   1:  PR[GP1:91,1] = PR[GP1:90,1] + 21.012;
   1:  PR[GP1:91,2] = PR[GP1:90,2] + -18.046;
   1:L PR[91] 10mm/sec CNT100;
   1:  PR[GP1:91,1] = PR[GP1:90,1] + 21.989;
   1:  PR[GP1:91,2] = PR[GP1:90,2] + -17.133;
   1:L PR[91] 10mm/sec CNT100;
   1:  PR[GP1:91,1] = PR[GP1:90,1] + 23.164;
   1:  PR[GP1:91,2] = PR[GP1:90,2] + -15.934;
   1:L PR[91] 10mm/sec CNT100;
   1:  PR[GP1:91,1] = PR[GP1:90,1] + 23.554;
   1:  PR[GP1:91,2] = PR[GP1:90,2] + -15.432;
   1:L PR[91] 10mm/sec CNT100;
   1:  PR[GP1:91,1] = PR[GP1:90,1] + 24.718;
   1:  PR[GP1:91,2] = PR[GP1:90,2] + -13.798;
   1:L PR[91] 10mm/sec CNT100;
   1:  PR[GP1:91,1] = PR[GP1:90,1] + 24.953;
   1:  PR[GP1:91,2] = PR[GP1:90,2] + -13.491;
   1:L PR[91] 10mm/sec CNT100;
   1:  PR[GP1:91,1] = PR[GP1:90,1] + 26.370;
   1:  PR[GP1:91,2] = PR[GP1:90,2] + -10.907;
   1:L PR[91] 10mm/sec CNT100;
   1:  PR[GP1:91,1] = PR[GP1:90,1] + 27.373;
   1:  PR[GP1:91,2] = PR[GP1:90,2] + -8.158;
   1:L PR[91] 10mm/sec CNT100;
   1:  PR[GP1:91,1] = PR[GP1:90,1] + 27.934;
   1:  PR[GP1:91,2] = PR[GP1:90,2] + -5.322;
   1:L PR[91] 10mm/sec CNT100;
   1:  PR[GP1:91,1] = PR[GP1:90,1] + 28.066;
   1:  PR[GP1:91,2] = PR[GP1:90,2] + -2.515;
   1:L PR[91] 10mm/sec CNT100;
   1:  PR[GP1:91,1] = PR[GP1:90,1] + 27.956;
   1:  PR[GP1:91,2] = PR[GP1:90,2] + -1.536;
   1:L PR[91] 10mm/sec CNT100;
   1:  PR[GP1:91,1] = PR[GP1:90,1] + 27.632;
   1:  PR[GP1:91,2] = PR[GP1:90,2] + 0.969;
   1:L PR[91] 10mm/sec CNT100;
   1:  PR[GP1:91,1] = PR[GP1:90,1] + 26.516;
   1:  PR[GP1:91,2] = PR[GP1:90,2] + 4.243;
   1:L PR[91] 10mm/sec CNT100;
   1:  PR[GP1:91,1] = PR[GP1:90,1] + 24.774;
   1:  PR[GP1:91,2] = PR[GP1:90,2] + 7.177;
   1:L PR[91] 10mm/sec CNT100;
   1:  PR[GP1:91,1] = PR[GP1:90,1] + 22.490;
   1:  PR[GP1:91,2] = PR[GP1:90,2] + 9.677;
   1:L PR[91] 10mm/sec CNT100;
   1:  PR[GP1:91,1] = PR[GP1:90,1] + 21.756;
   1:  PR[GP1:91,2] = PR[GP1:90,2] + 10.214;
   1:L PR[91] 10mm/sec CNT100;
   1:  PR[GP1:91,1] = PR[GP1:90,1] + 19.758;
   1:  PR[GP1:91,2] = PR[GP1:90,2] + 11.659;
   1:L PR[91] 10mm/sec CNT100;
   1:  PR[GP1:91,1] = PR[GP1:90,1] + 16.663;
   1:  PR[GP1:91,2] = PR[GP1:90,2] + 13.071;
   1:L PR[91] 10mm/sec CNT100;
   1:  PR[GP1:91,1] = PR[GP1:90,1] + 13.308;
   1:  PR[GP1:91,2] = PR[GP1:90,2] + 13.868;
   1:L PR[91] 10mm/sec CNT100;
   1:  PR[GP1:91,1] = PR[GP1:90,1] + 9.910;
   1:  PR[GP1:91,2] = PR[GP1:90,2] + 14.002;
   1:L PR[91] 10mm/sec CNT100;
   1:  PR[GP1:91,1] = PR[GP1:90,1] + 6.569;
   1:  PR[GP1:91,2] = PR[GP1:90,2] + 13.484;
   1:L PR[91] 10mm/sec CNT100;
   1:  PR[GP1:91,1] = PR[GP1:90,1] + 3.289;
   1:  PR[GP1:91,2] = PR[GP1:90,2] + 12.332;
   1:L PR[91] 10mm/sec CNT100;
   1:  PR[GP1:91,1] = PR[GP1:90,1] + 2.867;
   1:  PR[GP1:91,2] = PR[GP1:90,2] + 12.167;
   1:L PR[91] 10mm/sec CNT100;
   1:  PR[GP1:91,1] = PR[GP1:90,1] + 2.443;
   1:  PR[GP1:91,2] = PR[GP1:90,2] + 11.963;
   1:L PR[91] 10mm/sec CNT100;
   1:  PR[GP1:91,1] = PR[GP1:90,1] + 1.134;
   1:  PR[GP1:91,2] = PR[GP1:90,2] + 11.701;
   1:L PR[91] 10mm/sec CNT100;
   1:  PR[GP1:91,1] = PR[GP1:90,1] + 0.392;
   1:  PR[GP1:91,2] = PR[GP1:90,2] + 11.851;
   1:L PR[91] 10mm/sec CNT100;
   1:  PR[GP1:91,1] = PR[GP1:90,1] + -0.582;
   1:  PR[GP1:91,2] = PR[GP1:90,2] + 12.179;
   1:L PR[91] 10mm/sec CNT100;
   1:  PR[GP1:91,1] = PR[GP1:90,1] + -1.398;
   1:  PR[GP1:91,2] = PR[GP1:90,2] + 12.423;
   1:L PR[91] 10mm/sec CNT100;
   1:  PR[GP1:91,1] = PR[GP1:90,1] + -1.769;
   1:  PR[GP1:91,2] = PR[GP1:90,2] + 12.518;
   1:L PR[91] 10mm/sec CNT100;
   1:  PR[GP1:91,1] = PR[GP1:90,1] + -4.247;
   1:  PR[GP1:91,2] = PR[GP1:90,2] + 13.099;
   1:L PR[91] 10mm/sec CNT100;
   1:  PR[GP1:91,1] = PR[GP1:90,1] + -5.225;
   1:  PR[GP1:91,2] = PR[GP1:90,2] + 13.264;
   1:L PR[91] 10mm/sec CNT100;
   1:  PR[GP1:91,1] = PR[GP1:90,1] + -7.861;
   1:  PR[GP1:91,2] = PR[GP1:90,2] + 13.602;
   1:L PR[91] 10mm/sec CNT100;
   1:  PR[GP1:91,1] = PR[GP1:90,1] + -10.489;
   1:  PR[GP1:91,2] = PR[GP1:90,2] + 13.626;
   1:L PR[91] 10mm/sec CNT100;
   1:  PR[GP1:91,1] = PR[GP1:90,1] + -11.733;
   1:  PR[GP1:91,2] = PR[GP1:90,2] + 13.530;
   1:L PR[91] 10mm/sec CNT100;
   1:  PR[GP1:91,1] = PR[GP1:90,1] + -13.508;
   1:  PR[GP1:91,2] = PR[GP1:90,2] + 13.328;
   1:L PR[91] 10mm/sec CNT100;
   1:  PR[GP1:91,1] = PR[GP1:90,1] + -17.046;
   1:  PR[GP1:91,2] = PR[GP1:90,2] + 12.458;
   1:L PR[91] 10mm/sec CNT100;
   1:  PR[GP1:91,1] = PR[GP1:90,1] + -17.326;
   1:  PR[GP1:91,2] = PR[GP1:90,2] + 12.351;
   1:L PR[91] 10mm/sec CNT100;
   1:  PR[GP1:91,1] = PR[GP1:90,1] + -18.942;
   1:  PR[GP1:91,2] = PR[GP1:90,2] + 11.624;
   1:L PR[91] 10mm/sec CNT100;
   1:  PR[GP1:91,1] = PR[GP1:90,1] + -20.346;
   1:  PR[GP1:91,2] = PR[GP1:90,2] + 10.955;
   1:L PR[91] 10mm/sec CNT100;
   1:  PR[GP1:91,1] = PR[GP1:90,1] + -20.668;
   1:  PR[GP1:91,2] = PR[GP1:90,2] + 10.742;
   1:L PR[91] 10mm/sec CNT100;
   1:  PR[GP1:91,1] = PR[GP1:90,1] + -23.016;
   1:  PR[GP1:91,2] = PR[GP1:90,2] + 8.981;
   1:L PR[91] 10mm/sec CNT100;
   1:  PR[GP1:91,1] = PR[GP1:90,1] + -23.744;
   1:  PR[GP1:91,2] = PR[GP1:90,2] + 8.223;
   1:L PR[91] 10mm/sec CNT100;
   1:  PR[GP1:91,1] = PR[GP1:90,1] + -25.239;
   1:  PR[GP1:91,2] = PR[GP1:90,2] + 6.489;
   1:L PR[91] 10mm/sec CNT100;
   1:  PR[GP1:91,1] = PR[GP1:90,1] + -25.974;
   1:  PR[GP1:91,2] = PR[GP1:90,2] + 5.258;
   1:L PR[91] 10mm/sec CNT100;
   1:  PR[GP1:91,1] = PR[GP1:90,1] + -26.895;
   1:  PR[GP1:91,2] = PR[GP1:90,2] + 3.561;
   1:L PR[91] 10mm/sec CNT100;
   1:  PR[GP1:91,1] = PR[GP1:90,1] + -27.389;
   1:  PR[GP1:91,2] = PR[GP1:90,2] + 2.055;
   1:L PR[91] 10mm/sec CNT100;
   1:  PR[GP1:91,1] = PR[GP1:90,1] + -27.899;
   1:  PR[GP1:91,2] = PR[GP1:90,2] + 0.349;
   1:L PR[91] 10mm/sec CNT100;
   1:  PR[GP1:91,1] = PR[GP1:90,1] + -27.981;
   1:  PR[GP1:91,2] = PR[GP1:90,2] + -1.199;
   1:L PR[91] 10mm/sec CNT100;
   1:  PR[GP1:91,1] = PR[GP1:90,1] + -28.107;
   1:  PR[GP1:91,2] = PR[GP1:90,2] + -2.353;
   1:L PR[91] 10mm/sec CNT100;
   1:  PR[GP1:91,1] = PR[GP1:90,1] + -28.126;
   1:  PR[GP1:91,2] = PR[GP1:90,2] + -3.024;
   1:L PR[91] 10mm/sec CNT100;
   1:  PR[GP1:91,1] = PR[GP1:90,1] + -27.809;
   1:  PR[GP1:91,2] = PR[GP1:90,2] + -4.338;
   1:L PR[91] 10mm/sec CNT100;
   1:  PR[GP1:91,1] = PR[GP1:90,1] + -27.384;
   1:  PR[GP1:91,2] = PR[GP1:90,2] + -6.573;
   1:L PR[91] 10mm/sec CNT100;
   1:  PR[GP1:91,1] = PR[GP1:90,1] + -26.082;
   1:  PR[GP1:91,2] = PR[GP1:90,2] + -9.859;
   1:L PR[91] 10mm/sec CNT100;
   1:  PR[GP1:91,1] = PR[GP1:90,1] + -25.098;
   1:  PR[GP1:91,2] = PR[GP1:90,2] + -11.325;
   1:L PR[91] 10mm/sec CNT100;
   1:  PR[GP1:91,1] = PR[GP1:90,1] + -24.065;
   1:  PR[GP1:91,2] = PR[GP1:90,2] + -12.765;
   1:L PR[91] 10mm/sec CNT100;
   1:  PR[GP1:91,1] = PR[GP1:90,1] + -23.826;
   1:  PR[GP1:91,2] = PR[GP1:90,2] + -13.037;
   1:L PR[91] 10mm/sec CNT100;
   1:  PR[GP1:91,1] = PR[GP1:90,1] + -21.725;
   1:  PR[GP1:91,2] = PR[GP1:90,2] + -15.036;
   1:L PR[91] 10mm/sec CNT100;
   1:  PR[GP1:91,1] = PR[GP1:90,1] + -19.832;
   1:  PR[GP1:91,2] = PR[GP1:90,2] + -16.187;
   1:  PR[GP1:91,3] = PR[GP1:90,3] + 37.400;
   1:L PR[91] 10mm/sec CNT100;
   1:  PR[GP1:91,1] = PR[GP1:90,1] + -19.095;
   1:  PR[GP1:91,2] = PR[GP1:90,2] + -16.677;
   1:L PR[91] 10mm/sec CNT100;
   1:  PR[GP1:91,1] = PR[GP1:90,1] + -16.804;
   1:  PR[GP1:91,2] = PR[GP1:90,2] + -18.166;
   1:L PR[91] 10mm/sec CNT100;
   1:  PR[GP1:91,1] = PR[GP1:90,1] + -14.134;
   1:  PR[GP1:91,2] = PR[GP1:90,2] + -19.465;
   1:L PR[91] 10mm/sec CNT100;
   1:  PR[GP1:91,1] = PR[GP1:90,1] + -13.059;
   1:  PR[GP1:91,2] = PR[GP1:90,2] + -19.937;
   1:L PR[91] 10mm/sec CNT100;
   1:  PR[GP1:91,1] = PR[GP1:90,1] + -10.699;
   1:  PR[GP1:91,2] = PR[GP1:90,2] + -20.757;
   1:L PR[91] 10mm/sec CNT100;
   1:  PR[GP1:91,1] = PR[GP1:90,1] + -8.029;
   1:  PR[GP1:91,2] = PR[GP1:90,2] + -21.395;
   1:L PR[91] 10mm/sec CNT100;
   1:  PR[GP1:91,1] = PR[GP1:90,1] + -6.377;
   1:  PR[GP1:91,2] = PR[GP1:90,2] + -21.749;
   1:L PR[91] 10mm/sec CNT100;
   1:  PR[GP1:91,1] = PR[GP1:90,1] + -5.286;
   1:  PR[GP1:91,2] = PR[GP1:90,2] + -21.845;
   1:L PR[91] 10mm/sec CNT100;
   1:  PR[GP1:91,1] = PR[GP1:90,1] + -1.083;
   1:  PR[GP1:91,2] = PR[GP1:90,2] + -22.066;
   1:L PR[91] 10mm/sec CNT100;
   1:  PR[GP1:91,1] = PR[GP1:90,1] + -0.849;
   1:  PR[GP1:91,2] = PR[GP1:90,2] + -22.058;
   1:L PR[91] 10mm/sec CNT100;
   1:  PR[GP1:91,1] = PR[GP1:90,1] + 0.695;
   1:  PR[GP1:91,2] = PR[GP1:90,2] + -21.837;
   1:L PR[91] 10mm/sec CNT100;
   1:  PR[GP1:91,1] = PR[GP1:90,1] + 3.686;
   1:  PR[GP1:91,2] = PR[GP1:90,2] + -21.563;
   1:L PR[91] 10mm/sec CNT100;
   1:  PR[GP1:91,1] = PR[GP1:90,1] + 4.828;
   1:  PR[GP1:91,2] = PR[GP1:90,2] + -21.636;
   1:L PR[91] 10mm/sec CNT100;
   1:  PR[GP1:91,1] = PR[GP1:90,1] + 7.253;
   1:  PR[GP1:91,2] = PR[GP1:90,2] + -22.196;
   1:L PR[91] 10mm/sec CNT100;
   1:  PR[GP1:91,1] = PR[GP1:90,1] + 7.750;
   1:  PR[GP1:91,2] = PR[GP1:90,2] + -22.271;
   1:L PR[91] 10mm/sec CNT100;
   1:  PR[GP1:91,1] = PR[GP1:90,1] + 9.996;
   1:  PR[GP1:91,2] = PR[GP1:90,2] + -22.414;
   1:L PR[91] 10mm/sec CNT100;
   1:  PR[GP1:91,1] = PR[GP1:90,1] + 10.580;
   1:  PR[GP1:91,2] = PR[GP1:90,2] + -22.410;
   1:L PR[91] 10mm/sec CNT100;
   1:  PR[GP1:91,1] = PR[GP1:90,1] + 12.766;
   1:  PR[GP1:91,2] = PR[GP1:90,2] + -22.182;
   1:L PR[91] 10mm/sec CNT100;
   1:  PR[GP1:91,1] = PR[GP1:90,1] + 13.348;
   1:  PR[GP1:91,2] = PR[GP1:90,2] + -22.084;
   1:L PR[91] 10mm/sec CNT100;
   1:  PR[GP1:91,1] = PR[GP1:90,1] + 15.521;
   1:  PR[GP1:91,2] = PR[GP1:90,2] + -21.475;
   1:L PR[91] 10mm/sec CNT100;
   1:  PR[GP1:91,1] = PR[GP1:90,1] + 15.993;
   1:  PR[GP1:91,2] = PR[GP1:90,2] + -21.316;
   1:L PR[91] 10mm/sec CNT100;
   1:  PR[GP1:91,1] = PR[GP1:90,1] + 18.220;
   1:  PR[GP1:91,2] = PR[GP1:90,2] + -20.263;
   1:L PR[91] 10mm/sec CNT100;
   1:  PR[GP1:91,1] = PR[GP1:90,1] + 18.464;
   1:  PR[GP1:91,2] = PR[GP1:90,2] + -20.135;
   1:L PR[91] 10mm/sec CNT100;
   1:  PR[GP1:91,1] = PR[GP1:90,1] + 20.758;
   1:  PR[GP1:91,2] = PR[GP1:90,2] + -18.540;
   1:L PR[91] 10mm/sec CNT100;
   1:  PR[GP1:91,1] = PR[GP1:90,1] + 22.565;
   1:  PR[GP1:91,2] = PR[GP1:90,2] + -16.852;
   1:L PR[91] 10mm/sec CNT100;
   1:  PR[GP1:91,1] = PR[GP1:90,1] + 22.942;
   1:  PR[GP1:91,2] = PR[GP1:90,2] + -16.467;
   1:L PR[91] 10mm/sec CNT100;
   1:  PR[GP1:91,1] = PR[GP1:90,1] + 24.069;
   1:  PR[GP1:91,2] = PR[GP1:90,2] + -15.016;
   1:L PR[91] 10mm/sec CNT100;
   1:  PR[GP1:91,1] = PR[GP1:90,1] + 24.767;
   1:  PR[GP1:91,2] = PR[GP1:90,2] + -14.036;
   1:L PR[91] 10mm/sec CNT100;
   1:  PR[GP1:91,1] = PR[GP1:90,1] + 25.287;
   1:  PR[GP1:91,2] = PR[GP1:90,2] + -13.094;
   1:L PR[91] 10mm/sec CNT100;
   1:  PR[GP1:91,1] = PR[GP1:90,1] + 26.166;
   1:  PR[GP1:91,2] = PR[GP1:90,2] + -11.348;
   1:L PR[91] 10mm/sec CNT100;
   1:  PR[GP1:91,1] = PR[GP1:90,1] + 26.521;
   1:  PR[GP1:91,2] = PR[GP1:90,2] + -10.307;
   1:L PR[91] 10mm/sec CNT100;
   1:  PR[GP1:91,1] = PR[GP1:90,1] + 27.176;
   1:  PR[GP1:91,2] = PR[GP1:90,2] + -8.541;
   1:L PR[91] 10mm/sec CNT100;
   1:  PR[GP1:91,1] = PR[GP1:90,1] + 27.757;
   1:  PR[GP1:91,2] = PR[GP1:90,2] + -5.709;
   1:L PR[91] 10mm/sec CNT100;
   1:  PR[GP1:91,1] = PR[GP1:90,1] + 27.820;
   1:  PR[GP1:91,2] = PR[GP1:90,2] + -3.864;
   1:L PR[91] 10mm/sec CNT100;
   1:  PR[GP1:91,1] = PR[GP1:90,1] + 27.835;
   1:  PR[GP1:91,2] = PR[GP1:90,2] + -2.835;
   1:L PR[91] 10mm/sec CNT100;
   1:  PR[GP1:91,1] = PR[GP1:90,1] + 27.396;
   1:  PR[GP1:91,2] = PR[GP1:90,2] + 0.695;
   1:L PR[91] 10mm/sec CNT100;
   1:  PR[GP1:91,1] = PR[GP1:90,1] + 26.293;
   1:  PR[GP1:91,2] = PR[GP1:90,2] + 3.983;
   1:L PR[91] 10mm/sec CNT100;
   1:  PR[GP1:91,1] = PR[GP1:90,1] + 24.552;
   1:  PR[GP1:91,2] = PR[GP1:90,2] + 6.933;
   1:L PR[91] 10mm/sec CNT100;
   1:  PR[GP1:91,1] = PR[GP1:90,1] + 22.263;
   1:  PR[GP1:91,2] = PR[GP1:90,2] + 9.449;
   1:L PR[91] 10mm/sec CNT100;
   1:  PR[GP1:91,1] = PR[GP1:90,1] + 20.511;
   1:  PR[GP1:91,2] = PR[GP1:90,2] + 10.732;
   1:L PR[91] 10mm/sec CNT100;
   1:  PR[GP1:91,1] = PR[GP1:90,1] + 19.522;
   1:  PR[GP1:91,2] = PR[GP1:90,2] + 11.448;
   1:L PR[91] 10mm/sec CNT100;
   1:  PR[GP1:91,1] = PR[GP1:90,1] + 16.409;
   1:  PR[GP1:91,2] = PR[GP1:90,2] + 12.874;
   1:L PR[91] 10mm/sec CNT100;
   1:  PR[GP1:91,1] = PR[GP1:90,1] + 13.155;
   1:  PR[GP1:91,2] = PR[GP1:90,2] + 13.652;
   1:L PR[91] 10mm/sec CNT100;
   1:  PR[GP1:91,1] = PR[GP1:90,1] + 9.719;
   1:  PR[GP1:91,2] = PR[GP1:90,2] + 13.804;
   1:L PR[91] 10mm/sec CNT100;
   1:  PR[GP1:91,1] = PR[GP1:90,1] + 9.011;
   1:  PR[GP1:91,2] = PR[GP1:90,2] + 13.706;
   1:L PR[91] 10mm/sec CNT100;
   1:  PR[GP1:91,1] = PR[GP1:90,1] + 6.398;
   1:  PR[GP1:91,2] = PR[GP1:90,2] + 13.292;
   1:L PR[91] 10mm/sec CNT100;
   1:  PR[GP1:91,1] = PR[GP1:90,1] + 3.118;
   1:  PR[GP1:91,2] = PR[GP1:90,2] + 12.148;
   1:L PR[91] 10mm/sec CNT100;
   1:  PR[GP1:91,1] = PR[GP1:90,1] + 2.622;
   1:  PR[GP1:91,2] = PR[GP1:90,2] + 11.953;
   1:L PR[91] 10mm/sec CNT100;
   1:  PR[GP1:91,1] = PR[GP1:90,1] + 1.327;
   1:  PR[GP1:91,2] = PR[GP1:90,2] + 11.705;
   1:L PR[91] 10mm/sec CNT100;
   1:  PR[GP1:91,1] = PR[GP1:90,1] + 0.669;
   1:  PR[GP1:91,2] = PR[GP1:90,2] + 11.858;
   1:L PR[91] 10mm/sec CNT100;
   1:  PR[GP1:91,1] = PR[GP1:90,1] + -0.435;
   1:  PR[GP1:91,2] = PR[GP1:90,2] + 12.188;
   1:L PR[91] 10mm/sec CNT100;
   1:  PR[GP1:91,1] = PR[GP1:90,1] + -0.928;
   1:  PR[GP1:91,2] = PR[GP1:90,2] + 12.315;
   1:L PR[91] 10mm/sec CNT100;
   1:  PR[GP1:91,1] = PR[GP1:90,1] + -2.534;
   1:  PR[GP1:91,2] = PR[GP1:90,2] + 12.694;
   1:L PR[91] 10mm/sec CNT100;
   1:  PR[GP1:91,1] = PR[GP1:90,1] + -3.060;
   1:  PR[GP1:91,2] = PR[GP1:90,2] + 12.812;
   1:L PR[91] 10mm/sec CNT100;
   1:  PR[GP1:91,1] = PR[GP1:90,1] + -4.631;
   1:  PR[GP1:91,2] = PR[GP1:90,2] + 13.077;
   1:L PR[91] 10mm/sec CNT100;
   1:  PR[GP1:91,1] = PR[GP1:90,1] + -6.914;
   1:  PR[GP1:91,2] = PR[GP1:90,2] + 13.369;
   1:L PR[91] 10mm/sec CNT100;
   1:  PR[GP1:91,1] = PR[GP1:90,1] + -10.028;
   1:  PR[GP1:91,2] = PR[GP1:90,2] + 13.428;
   1:L PR[91] 10mm/sec CNT100;
   1:  PR[GP1:91,1] = PR[GP1:90,1] + -12.823;
   1:  PR[GP1:91,2] = PR[GP1:90,2] + 13.118;
   1:L PR[91] 10mm/sec CNT100;
   1:  PR[GP1:91,1] = PR[GP1:90,1] + -16.123;
   1:  PR[GP1:91,2] = PR[GP1:90,2] + 12.304;
   1:L PR[91] 10mm/sec CNT100;
   1:  PR[GP1:91,1] = PR[GP1:90,1] + -16.912;
   1:  PR[GP1:91,2] = PR[GP1:90,2] + 12.003;
   1:L PR[91] 10mm/sec CNT100;
   1:  PR[GP1:91,1] = PR[GP1:90,1] + -19.663;
   1:  PR[GP1:91,2] = PR[GP1:90,2] + 10.766;
   1:L PR[91] 10mm/sec CNT100;
   1:  PR[GP1:91,1] = PR[GP1:90,1] + -19.823;
   1:  PR[GP1:91,2] = PR[GP1:90,2] + 10.679;
   1:L PR[91] 10mm/sec CNT100;
   1:  PR[GP1:91,1] = PR[GP1:90,1] + -20.996;
   1:  PR[GP1:91,2] = PR[GP1:90,2] + 9.844;
   1:L PR[91] 10mm/sec CNT100;
   1:  PR[GP1:91,1] = PR[GP1:90,1] + -22.533;
   1:  PR[GP1:91,2] = PR[GP1:90,2] + 8.692;
   1:L PR[91] 10mm/sec CNT100;
   1:  PR[GP1:91,1] = PR[GP1:90,1] + -22.765;
   1:  PR[GP1:91,2] = PR[GP1:90,2] + 8.450;
   1:L PR[91] 10mm/sec CNT100;
   1:  PR[GP1:91,1] = PR[GP1:90,1] + -24.701;
   1:  PR[GP1:91,2] = PR[GP1:90,2] + 6.205;
   1:L PR[91] 10mm/sec CNT100;
   1:  PR[GP1:91,1] = PR[GP1:90,1] + -25.091;
   1:  PR[GP1:91,2] = PR[GP1:90,2] + 5.551;
   1:L PR[91] 10mm/sec CNT100;
   1:  PR[GP1:91,1] = PR[GP1:90,1] + -26.314;
   1:  PR[GP1:91,2] = PR[GP1:90,2] + 3.296;
   1:L PR[91] 10mm/sec CNT100;
   1:  PR[GP1:91,1] = PR[GP1:90,1] + -26.610;
   1:  PR[GP1:91,2] = PR[GP1:90,2] + 2.395;
   1:L PR[91] 10mm/sec CNT100;
   1:  PR[GP1:91,1] = PR[GP1:90,1] + -27.292;
   1:  PR[GP1:91,2] = PR[GP1:90,2] + 0.114;
   1:L PR[91] 10mm/sec CNT100;
   1:  PR[GP1:91,1] = PR[GP1:90,1] + -27.342;
   1:  PR[GP1:91,2] = PR[GP1:90,2] + -0.825;
   1:L PR[91] 10mm/sec CNT100;
   1:  PR[GP1:91,1] = PR[GP1:90,1] + -27.420;
   1:  PR[GP1:91,2] = PR[GP1:90,2] + -1.538;
   1:L PR[91] 10mm/sec CNT100;
   1:  PR[GP1:91,1] = PR[GP1:90,1] + -27.467;
   1:  PR[GP1:91,2] = PR[GP1:90,2] + -3.238;
   1:L PR[91] 10mm/sec CNT100;
   1:  PR[GP1:91,1] = PR[GP1:90,1] + -27.297;
   1:  PR[GP1:91,2] = PR[GP1:90,2] + -3.942;
   1:L PR[91] 10mm/sec CNT100;
   1:  PR[GP1:91,1] = PR[GP1:90,1] + -26.763;
   1:  PR[GP1:91,2] = PR[GP1:90,2] + -6.745;
   1:L PR[91] 10mm/sec CNT100;
   1:  PR[GP1:91,1] = PR[GP1:90,1] + -25.976;
   1:  PR[GP1:91,2] = PR[GP1:90,2] + -8.742;
   1:L PR[91] 10mm/sec CNT100;
   1:  PR[GP1:91,1] = PR[GP1:90,1] + -25.440;
   1:  PR[GP1:91,2] = PR[GP1:90,2] + -9.977;
   1:L PR[91] 10mm/sec CNT100;
   1:  PR[GP1:91,1] = PR[GP1:90,1] + -25.345;
   1:  PR[GP1:91,2] = PR[GP1:90,2] + -10.127;
   1:L PR[91] 10mm/sec CNT100;
   1:  PR[GP1:91,1] = PR[GP1:90,1] + -23.474;
   1:  PR[GP1:91,2] = PR[GP1:90,2] + -12.733;
   1:L PR[91] 10mm/sec CNT100;
   1:  PR[GP1:91,1] = PR[GP1:90,1] + -22.802;
   1:  PR[GP1:91,2] = PR[GP1:90,2] + -13.499;
   1:L PR[91] 10mm/sec CNT100;
   1:  PR[GP1:91,1] = PR[GP1:90,1] + -21.280;
   1:  PR[GP1:91,2] = PR[GP1:90,2] + -14.947;
   1:L PR[91] 10mm/sec CNT100;
   1:  PR[GP1:91,1] = PR[GP1:90,1] + -18.916;
   1:  PR[GP1:91,2] = PR[GP1:90,2] + -16.501;
   1:  PR[GP1:91,3] = PR[GP1:90,3] + 38.500;
   1:L PR[91] 10mm/sec CNT100;
   1:  PR[GP1:91,1] = PR[GP1:90,1] + -15.891;
   1:  PR[GP1:91,2] = PR[GP1:90,2] + -18.471;
   1:L PR[91] 10mm/sec CNT100;
   1:  PR[GP1:91,1] = PR[GP1:90,1] + -13.552;
   1:  PR[GP1:91,2] = PR[GP1:90,2] + -19.609;
   1:L PR[91] 10mm/sec CNT100;
   1:  PR[GP1:91,1] = PR[GP1:90,1] + -11.911;
   1:  PR[GP1:91,2] = PR[GP1:90,2] + -20.329;
   1:L PR[91] 10mm/sec CNT100;
   1:  PR[GP1:91,1] = PR[GP1:90,1] + -9.976;
   1:  PR[GP1:91,2] = PR[GP1:90,2] + -21.001;
   1:L PR[91] 10mm/sec CNT100;
   1:  PR[GP1:91,1] = PR[GP1:90,1] + -6.564;
   1:  PR[GP1:91,2] = PR[GP1:90,2] + -21.817;
   1:L PR[91] 10mm/sec CNT100;
   1:  PR[GP1:91,1] = PR[GP1:90,1] + -5.457;
   1:  PR[GP1:91,2] = PR[GP1:90,2] + -22.054;
   1:L PR[91] 10mm/sec CNT100;
   1:  PR[GP1:91,1] = PR[GP1:90,1] + -4.733;
   1:  PR[GP1:91,2] = PR[GP1:90,2] + -22.118;
   1:L PR[91] 10mm/sec CNT100;
   1:  PR[GP1:91,1] = PR[GP1:90,1] + -0.660;
   1:  PR[GP1:91,2] = PR[GP1:90,2] + -22.332;
   1:L PR[91] 10mm/sec CNT100;
   1:  PR[GP1:91,1] = PR[GP1:90,1] + 0.067;
   1:  PR[GP1:91,2] = PR[GP1:90,2] + -22.399;
   1:L PR[91] 10mm/sec CNT100;
   1:  PR[GP1:91,1] = PR[GP1:90,1] + 4.181;
   1:  PR[GP1:91,2] = PR[GP1:90,2] + -22.017;
   1:L PR[91] 10mm/sec CNT100;
   1:  PR[GP1:91,1] = PR[GP1:90,1] + 5.247;
   1:  PR[GP1:91,2] = PR[GP1:90,2] + -22.084;
   1:L PR[91] 10mm/sec CNT100;
   1:  PR[GP1:91,1] = PR[GP1:90,1] + 6.980;
   1:  PR[GP1:91,2] = PR[GP1:90,2] + -22.475;
   1:L PR[91] 10mm/sec CNT100;
   1:  PR[GP1:91,1] = PR[GP1:90,1] + 8.189;
   1:  PR[GP1:91,2] = PR[GP1:90,2] + -22.656;
   1:L PR[91] 10mm/sec CNT100;
   1:  PR[GP1:91,1] = PR[GP1:90,1] + 9.649;
   1:  PR[GP1:91,2] = PR[GP1:90,2] + -22.750;
   1:L PR[91] 10mm/sec CNT100;
   1:  PR[GP1:91,1] = PR[GP1:90,1] + 11.005;
   1:  PR[GP1:91,2] = PR[GP1:90,2] + -22.739;
   1:L PR[91] 10mm/sec CNT100;
   1:  PR[GP1:91,1] = PR[GP1:90,1] + 12.338;
   1:  PR[GP1:91,2] = PR[GP1:90,2] + -22.600;
   1:L PR[91] 10mm/sec CNT100;
   1:  PR[GP1:91,1] = PR[GP1:90,1] + 13.748;
   1:  PR[GP1:91,2] = PR[GP1:90,2] + -22.364;
   1:L PR[91] 10mm/sec CNT100;
   1:  PR[GP1:91,1] = PR[GP1:90,1] + 15.010;
   1:  PR[GP1:91,2] = PR[GP1:90,2] + -22.010;
   1:L PR[91] 10mm/sec CNT100;
   1:  PR[GP1:91,1] = PR[GP1:90,1] + 16.359;
   1:  PR[GP1:91,2] = PR[GP1:90,2] + -21.556;
   1:L PR[91] 10mm/sec CNT100;
   1:  PR[GP1:91,1] = PR[GP1:90,1] + 17.629;
   1:  PR[GP1:91,2] = PR[GP1:90,2] + -20.956;
   1:L PR[91] 10mm/sec CNT100;
   1:  PR[GP1:91,1] = PR[GP1:90,1] + 18.786;
   1:  PR[GP1:91,2] = PR[GP1:90,2] + -20.350;
   1:L PR[91] 10mm/sec CNT100;
   1:  PR[GP1:91,1] = PR[GP1:90,1] + 20.151;
   1:  PR[GP1:91,2] = PR[GP1:90,2] + -19.396;
   1:L PR[91] 10mm/sec CNT100;
   1:  PR[GP1:91,1] = PR[GP1:90,1] + 20.988;
   1:  PR[GP1:91,2] = PR[GP1:90,2] + -18.773;
   1:L PR[91] 10mm/sec CNT100;
   1:  PR[GP1:91,1] = PR[GP1:90,1] + 22.521;
   1:  PR[GP1:91,2] = PR[GP1:90,2] + -17.270;
   1:L PR[91] 10mm/sec CNT100;
   1:  PR[GP1:91,1] = PR[GP1:90,1] + 22.928;
   1:  PR[GP1:91,2] = PR[GP1:90,2] + -16.854;
   1:L PR[91] 10mm/sec CNT100;
   1:  PR[GP1:91,1] = PR[GP1:90,1] + 24.594;
   1:  PR[GP1:91,2] = PR[GP1:90,2] + -14.584;
   1:L PR[91] 10mm/sec CNT100;
   1:  PR[GP1:91,1] = PR[GP1:90,1] + 25.711;
   1:  PR[GP1:91,2] = PR[GP1:90,2] + -12.559;
   1:L PR[91] 10mm/sec CNT100;
   1:  PR[GP1:91,1] = PR[GP1:90,1] + 26.045;
   1:  PR[GP1:91,2] = PR[GP1:90,2] + -11.895;
   1:L PR[91] 10mm/sec CNT100;
   1:  PR[GP1:91,1] = PR[GP1:90,1] + 26.567;
   1:  PR[GP1:91,2] = PR[GP1:90,2] + -10.480;
   1:L PR[91] 10mm/sec CNT100;
   1:  PR[GP1:91,1] = PR[GP1:90,1] + 27.047;
   1:  PR[GP1:91,2] = PR[GP1:90,2] + -9.029;
   1:L PR[91] 10mm/sec CNT100;
   1:  PR[GP1:91,1] = PR[GP1:90,1] + 27.183;
   1:  PR[GP1:91,2] = PR[GP1:90,2] + -8.364;
   1:L PR[91] 10mm/sec CNT100;
   1:  PR[GP1:91,1] = PR[GP1:90,1] + 27.582;
   1:  PR[GP1:91,2] = PR[GP1:90,2] + -6.102;
   1:L PR[91] 10mm/sec CNT100;
   1:  PR[GP1:91,1] = PR[GP1:90,1] + 27.694;
   1:  PR[GP1:91,2] = PR[GP1:90,2] + -3.225;
   1:L PR[91] 10mm/sec CNT100;
   1:  PR[GP1:91,1] = PR[GP1:90,1] + 27.195;
   1:  PR[GP1:91,2] = PR[GP1:90,2] + 0.389;
   1:L PR[91] 10mm/sec CNT100;
   1:  PR[GP1:91,1] = PR[GP1:90,1] + 26.701;
   1:  PR[GP1:91,2] = PR[GP1:90,2] + 1.818;
   1:L PR[91] 10mm/sec CNT100;
   1:  PR[GP1:91,1] = PR[GP1:90,1] + 26.070;
   1:  PR[GP1:91,2] = PR[GP1:90,2] + 3.722;
   1:L PR[91] 10mm/sec CNT100;
   1:  PR[GP1:91,1] = PR[GP1:90,1] + 24.330;
   1:  PR[GP1:91,2] = PR[GP1:90,2] + 6.689;
   1:L PR[91] 10mm/sec CNT100;
   1:  PR[GP1:91,1] = PR[GP1:90,1] + 22.035;
   1:  PR[GP1:91,2] = PR[GP1:90,2] + 9.222;
   1:L PR[91] 10mm/sec CNT100;
   1:  PR[GP1:91,1] = PR[GP1:90,1] + 19.282;
   1:  PR[GP1:91,2] = PR[GP1:90,2] + 11.237;
   1:L PR[91] 10mm/sec CNT100;
   1:  PR[GP1:91,1] = PR[GP1:90,1] + 16.261;
   1:  PR[GP1:91,2] = PR[GP1:90,2] + 12.645;
   1:L PR[91] 10mm/sec CNT100;
   1:  PR[GP1:91,1] = PR[GP1:90,1] + 13.003;
   1:  PR[GP1:91,2] = PR[GP1:90,2] + 13.436;
   1:L PR[91] 10mm/sec CNT100;
   1:  PR[GP1:91,1] = PR[GP1:90,1] + 9.620;
   1:  PR[GP1:91,2] = PR[GP1:90,2] + 13.586;
   1:L PR[91] 10mm/sec CNT100;
   1:  PR[GP1:91,1] = PR[GP1:90,1] + 7.086;
   1:  PR[GP1:91,2] = PR[GP1:90,2] + 13.236;
   1:L PR[91] 10mm/sec CNT100;
   1:  PR[GP1:91,1] = PR[GP1:90,1] + 6.226;
   1:  PR[GP1:91,2] = PR[GP1:90,2] + 13.099;
   1:L PR[91] 10mm/sec CNT100;
   1:  PR[GP1:91,1] = PR[GP1:90,1] + 2.820;
   1:  PR[GP1:91,2] = PR[GP1:90,2] + 11.916;
   1:L PR[91] 10mm/sec CNT100;
   1:  PR[GP1:91,1] = PR[GP1:90,1] + 1.538;
   1:  PR[GP1:91,2] = PR[GP1:90,2] + 11.705;
   1:L PR[91] 10mm/sec CNT100;
   1:  PR[GP1:91,1] = PR[GP1:90,1] + 0.971;
   1:  PR[GP1:91,2] = PR[GP1:90,2] + 11.821;
   1:L PR[91] 10mm/sec CNT100;
   1:  PR[GP1:91,1] = PR[GP1:90,1] + 0.528;
   1:  PR[GP1:91,2] = PR[GP1:90,2] + 11.954;
   1:L PR[91] 10mm/sec CNT100;
   1:  PR[GP1:91,1] = PR[GP1:90,1] + -0.085;
   1:  PR[GP1:91,2] = PR[GP1:90,2] + 12.112;
   1:L PR[91] 10mm/sec CNT100;
   1:  PR[GP1:91,1] = PR[GP1:90,1] + -1.879;
   1:  PR[GP1:91,2] = PR[GP1:90,2] + 12.527;
   1:L PR[91] 10mm/sec CNT100;
   1:  PR[GP1:91,1] = PR[GP1:90,1] + -4.037;
   1:  PR[GP1:91,2] = PR[GP1:90,2] + 12.890;
   1:L PR[91] 10mm/sec CNT100;
   1:  PR[GP1:91,1] = PR[GP1:90,1] + -5.962;
   1:  PR[GP1:91,2] = PR[GP1:90,2] + 13.137;
   1:L PR[91] 10mm/sec CNT100;
   1:  PR[GP1:91,1] = PR[GP1:90,1] + -9.327;
   1:  PR[GP1:91,2] = PR[GP1:90,2] + 13.196;
   1:L PR[91] 10mm/sec CNT100;
   1:  PR[GP1:91,1] = PR[GP1:90,1] + -11.088;
   1:  PR[GP1:91,2] = PR[GP1:90,2] + 13.026;
   1:L PR[91] 10mm/sec CNT100;
   1:  PR[GP1:91,1] = PR[GP1:90,1] + -12.136;
   1:  PR[GP1:91,2] = PR[GP1:90,2] + 12.908;
   1:L PR[91] 10mm/sec CNT100;
   1:  PR[GP1:91,1] = PR[GP1:90,1] + -15.201;
   1:  PR[GP1:91,2] = PR[GP1:90,2] + 12.151;
   1:L PR[91] 10mm/sec CNT100;
   1:  PR[GP1:91,1] = PR[GP1:90,1] + -16.498;
   1:  PR[GP1:91,2] = PR[GP1:90,2] + 11.656;
   1:L PR[91] 10mm/sec CNT100;
   1:  PR[GP1:91,1] = PR[GP1:90,1] + -18.532;
   1:  PR[GP1:91,2] = PR[GP1:90,2] + 10.741;
   1:L PR[91] 10mm/sec CNT100;
   1:  PR[GP1:91,1] = PR[GP1:90,1] + -19.213;
   1:  PR[GP1:91,2] = PR[GP1:90,2] + 10.369;
   1:L PR[91] 10mm/sec CNT100;
   1:  PR[GP1:91,1] = PR[GP1:90,1] + -21.917;
   1:  PR[GP1:91,2] = PR[GP1:90,2] + 8.438;
   1:L PR[91] 10mm/sec CNT100;
   1:  PR[GP1:91,1] = PR[GP1:90,1] + -23.406;
   1:  PR[GP1:91,2] = PR[GP1:90,2] + 6.799;
   1:L PR[91] 10mm/sec CNT100;
   1:  PR[GP1:91,1] = PR[GP1:90,1] + -24.162;
   1:  PR[GP1:91,2] = PR[GP1:90,2] + 5.922;
   1:L PR[91] 10mm/sec CNT100;
   1:  PR[GP1:91,1] = PR[GP1:90,1] + -24.209;
   1:  PR[GP1:91,2] = PR[GP1:90,2] + 5.844;
   1:L PR[91] 10mm/sec CNT100;
   1:  PR[GP1:91,1] = PR[GP1:90,1] + -25.730;
   1:  PR[GP1:91,2] = PR[GP1:90,2] + 3.038;
   1:L PR[91] 10mm/sec CNT100;
   1:  PR[GP1:91,1] = PR[GP1:90,1] + -26.688;
   1:  PR[GP1:91,2] = PR[GP1:90,2] + -0.131;
   1:L PR[91] 10mm/sec CNT100;
   1:  PR[GP1:91,1] = PR[GP1:90,1] + -26.732;
   1:  PR[GP1:91,2] = PR[GP1:90,2] + -0.713;
   1:L PR[91] 10mm/sec CNT100;
   1:  PR[GP1:91,1] = PR[GP1:90,1] + -26.807;
   1:  PR[GP1:91,2] = PR[GP1:90,2] + -3.452;
   1:L PR[91] 10mm/sec CNT100;
   1:  PR[GP1:91,1] = PR[GP1:90,1] + -26.785;
   1:  PR[GP1:91,2] = PR[GP1:90,2] + -3.546;
   1:L PR[91] 10mm/sec CNT100;
   1:  PR[GP1:91,1] = PR[GP1:90,1] + -26.546;
   1:  PR[GP1:91,2] = PR[GP1:90,2] + -4.800;
   1:L PR[91] 10mm/sec CNT100;
   1:  PR[GP1:91,1] = PR[GP1:90,1] + -26.118;
   1:  PR[GP1:91,2] = PR[GP1:90,2] + -6.738;
   1:L PR[91] 10mm/sec CNT100;
   1:  PR[GP1:91,1] = PR[GP1:90,1] + -26.078;
   1:  PR[GP1:91,2] = PR[GP1:90,2] + -6.912;
   1:L PR[91] 10mm/sec CNT100;
   1:  PR[GP1:91,1] = PR[GP1:90,1] + -25.995;
   1:  PR[GP1:91,2] = PR[GP1:90,2] + -7.118;
   1:L PR[91] 10mm/sec CNT100;
   1:  PR[GP1:91,1] = PR[GP1:90,1] + -24.719;
   1:  PR[GP1:91,2] = PR[GP1:90,2] + -10.057;
   1:L PR[91] 10mm/sec CNT100;
   1:  PR[GP1:91,1] = PR[GP1:90,1] + -24.274;
   1:  PR[GP1:91,2] = PR[GP1:90,2] + -10.764;
   1:L PR[91] 10mm/sec CNT100;
   1:  PR[GP1:91,1] = PR[GP1:90,1] + -22.883;
   1:  PR[GP1:91,2] = PR[GP1:90,2] + -12.701;
   1:L PR[91] 10mm/sec CNT100;
   1:  PR[GP1:91,1] = PR[GP1:90,1] + -21.778;
   1:  PR[GP1:91,2] = PR[GP1:90,2] + -13.961;
   1:L PR[91] 10mm/sec CNT100;
   1:  PR[GP1:91,1] = PR[GP1:90,1] + -20.834;
   1:  PR[GP1:91,2] = PR[GP1:90,2] + -14.858;
   1:L PR[91] 10mm/sec CNT100;
   1:  PR[GP1:91,1] = PR[GP1:90,1] + -20.389;
   1:  PR[GP1:91,2] = PR[GP1:90,2] + -14.770;
   1:  PR[GP1:91,3] = PR[GP1:90,3] + 39.600;
   1:L PR[91] 10mm/sec CNT100;
   1:  PR[GP1:91,1] = PR[GP1:90,1] + -18.113;
   1:  PR[GP1:91,2] = PR[GP1:90,2] + -16.722;
   1:L PR[91] 10mm/sec CNT100;
   1:  PR[GP1:91,1] = PR[GP1:90,1] + -17.695;
   1:  PR[GP1:91,2] = PR[GP1:90,2] + -17.008;
   1:L PR[91] 10mm/sec CNT100;
   1:  PR[GP1:91,1] = PR[GP1:90,1] + -14.979;
   1:  PR[GP1:91,2] = PR[GP1:90,2] + -18.775;
   1:L PR[91] 10mm/sec CNT100;
   1:  PR[GP1:91,1] = PR[GP1:90,1] + -12.969;
   1:  PR[GP1:91,2] = PR[GP1:90,2] + -19.753;
   1:L PR[91] 10mm/sec CNT100;
   1:  PR[GP1:91,1] = PR[GP1:90,1] + -10.762;
   1:  PR[GP1:91,2] = PR[GP1:90,2] + -20.721;
   1:L PR[91] 10mm/sec CNT100;
   1:  PR[GP1:91,1] = PR[GP1:90,1] + -9.253;
   1:  PR[GP1:91,2] = PR[GP1:90,2] + -21.245;
   1:L PR[91] 10mm/sec CNT100;
   1:  PR[GP1:91,1] = PR[GP1:90,1] + -5.099;
   1:  PR[GP1:91,2] = PR[GP1:90,2] + -22.239;
   1:L PR[91] 10mm/sec CNT100;
   1:  PR[GP1:91,1] = PR[GP1:90,1] + -4.537;
   1:  PR[GP1:91,2] = PR[GP1:90,2] + -22.359;
   1:L PR[91] 10mm/sec CNT100;
   1:  PR[GP1:91,1] = PR[GP1:90,1] + -4.179;
   1:  PR[GP1:91,2] = PR[GP1:90,2] + -22.390;
   1:L PR[91] 10mm/sec CNT100;
   1:  PR[GP1:91,1] = PR[GP1:90,1] + -2.024;
   1:  PR[GP1:91,2] = PR[GP1:90,2] + -22.504;
   1:L PR[91] 10mm/sec CNT100;
   1:  PR[GP1:91,1] = PR[GP1:90,1] + 0.476;
   1:  PR[GP1:91,2] = PR[GP1:90,2] + -22.773;
   1:L PR[91] 10mm/sec CNT100;
   1:  PR[GP1:91,1] = PR[GP1:90,1] + 1.191;
   1:  PR[GP1:91,2] = PR[GP1:90,2] + -22.803;
   1:L PR[91] 10mm/sec CNT100;
   1:  PR[GP1:91,1] = PR[GP1:90,1] + 4.701;
   1:  PR[GP1:91,2] = PR[GP1:90,2] + -22.468;
   1:L PR[91] 10mm/sec CNT100;
   1:  PR[GP1:91,1] = PR[GP1:90,1] + 5.689;
   1:  PR[GP1:91,2] = PR[GP1:90,2] + -22.529;
   1:L PR[91] 10mm/sec CNT100;
   1:  PR[GP1:91,1] = PR[GP1:90,1] + 6.707;
   1:  PR[GP1:91,2] = PR[GP1:90,2] + -22.753;
   1:L PR[91] 10mm/sec CNT100;
   1:  PR[GP1:91,1] = PR[GP1:90,1] + 8.628;
   1:  PR[GP1:91,2] = PR[GP1:90,2] + -23.042;
   1:L PR[91] 10mm/sec CNT100;
   1:  PR[GP1:91,1] = PR[GP1:90,1] + 9.302;
   1:  PR[GP1:91,2] = PR[GP1:90,2] + -23.085;
   1:L PR[91] 10mm/sec CNT100;
   1:  PR[GP1:91,1] = PR[GP1:90,1] + 11.431;
   1:  PR[GP1:91,2] = PR[GP1:90,2] + -23.069;
   1:L PR[91] 10mm/sec CNT100;
   1:  PR[GP1:91,1] = PR[GP1:90,1] + 11.909;
   1:  PR[GP1:91,2] = PR[GP1:90,2] + -23.019;
   1:L PR[91] 10mm/sec CNT100;
   1:  PR[GP1:91,1] = PR[GP1:90,1] + 14.149;
   1:  PR[GP1:91,2] = PR[GP1:90,2] + -22.644;
   1:L PR[91] 10mm/sec CNT100;
   1:  PR[GP1:91,1] = PR[GP1:90,1] + 14.498;
   1:  PR[GP1:91,2] = PR[GP1:90,2] + -22.546;
   1:L PR[91] 10mm/sec CNT100;
   1:  PR[GP1:91,1] = PR[GP1:90,1] + 16.724;
   1:  PR[GP1:91,2] = PR[GP1:90,2] + -21.797;
   1:L PR[91] 10mm/sec CNT100;
   1:  PR[GP1:91,1] = PR[GP1:90,1] + 17.037;
   1:  PR[GP1:91,2] = PR[GP1:90,2] + -21.649;
   1:L PR[91] 10mm/sec CNT100;
   1:  PR[GP1:91,1] = PR[GP1:90,1] + 19.108;
   1:  PR[GP1:91,2] = PR[GP1:90,2] + -20.564;
   1:L PR[91] 10mm/sec CNT100;
   1:  PR[GP1:91,1] = PR[GP1:90,1] + 19.493;
   1:  PR[GP1:91,2] = PR[GP1:90,2] + -20.296;
   1:L PR[91] 10mm/sec CNT100;
   1:  PR[GP1:91,1] = PR[GP1:90,1] + 21.261;
   1:  PR[GP1:91,2] = PR[GP1:90,2] + -18.978;
   1:L PR[91] 10mm/sec CNT100;
   1:  PR[GP1:91,1] = PR[GP1:90,1] + 21.821;
   1:  PR[GP1:91,2] = PR[GP1:90,2] + -18.429;
   1:L PR[91] 10mm/sec CNT100;
   1:  PR[GP1:91,1] = PR[GP1:90,1] + 23.148;
   1:  PR[GP1:91,2] = PR[GP1:90,2] + -17.072;
   1:L PR[91] 10mm/sec CNT100;
   1:  PR[GP1:91,1] = PR[GP1:90,1] + 24.741;
   1:  PR[GP1:91,2] = PR[GP1:90,2] + -14.860;
   1:L PR[91] 10mm/sec CNT100;
   1:  PR[GP1:91,1] = PR[GP1:90,1] + 26.007;
   1:  PR[GP1:91,2] = PR[GP1:90,2] + -12.369;
   1:L PR[91] 10mm/sec CNT100;
   1:  PR[GP1:91,1] = PR[GP1:90,1] + 26.508;
   1:  PR[GP1:91,2] = PR[GP1:90,2] + -10.856;
   1:L PR[91] 10mm/sec CNT100;
   1:  PR[GP1:91,1] = PR[GP1:90,1] + 26.878;
   1:  PR[GP1:91,2] = PR[GP1:90,2] + -9.854;
   1:L PR[91] 10mm/sec CNT100;
   1:  PR[GP1:91,1] = PR[GP1:90,1] + 26.972;
   1:  PR[GP1:91,2] = PR[GP1:90,2] + -9.569;
   1:L PR[91] 10mm/sec CNT100;
   1:  PR[GP1:91,1] = PR[GP1:90,1] + 27.357;
   1:  PR[GP1:91,2] = PR[GP1:90,2] + -7.683;
   1:L PR[91] 10mm/sec CNT100;
   1:  PR[GP1:91,1] = PR[GP1:90,1] + 27.543;
   1:  PR[GP1:91,2] = PR[GP1:90,2] + -6.613;
   1:L PR[91] 10mm/sec CNT100;
   1:  PR[GP1:91,1] = PR[GP1:90,1] + 27.604;
   1:  PR[GP1:91,2] = PR[GP1:90,2] + -3.657;
   1:L PR[91] 10mm/sec CNT100;
   1:  PR[GP1:91,1] = PR[GP1:90,1] + 27.454;
   1:  PR[GP1:91,2] = PR[GP1:90,2] + -2.655;
   1:L PR[91] 10mm/sec CNT100;
   1:  PR[GP1:91,1] = PR[GP1:90,1] + 27.109;
   1:  PR[GP1:91,2] = PR[GP1:90,2] + 0.004;
   1:L PR[91] 10mm/sec CNT100;
   1:  PR[GP1:91,1] = PR[GP1:90,1] + 26.463;
   1:  PR[GP1:91,2] = PR[GP1:90,2] + 1.876;
   1:L PR[91] 10mm/sec CNT100;
   1:  PR[GP1:91,1] = PR[GP1:90,1] + 25.962;
   1:  PR[GP1:91,2] = PR[GP1:90,2] + 3.394;
   1:L PR[91] 10mm/sec CNT100;
   1:  PR[GP1:91,1] = PR[GP1:90,1] + 25.530;
   1:  PR[GP1:91,2] = PR[GP1:90,2] + 4.150;
   1:L PR[91] 10mm/sec CNT100;
   1:  PR[GP1:91,1] = PR[GP1:90,1] + 24.196;
   1:  PR[GP1:91,2] = PR[GP1:90,2] + 6.402;
   1:L PR[91] 10mm/sec CNT100;
   1:  PR[GP1:91,1] = PR[GP1:90,1] + 21.906;
   1:  PR[GP1:91,2] = PR[GP1:90,2] + 8.955;
   1:L PR[91] 10mm/sec CNT100;
   1:  PR[GP1:91,1] = PR[GP1:90,1] + 19.193;
   1:  PR[GP1:91,2] = PR[GP1:90,2] + 10.974;
   1:L PR[91] 10mm/sec CNT100;
   1:  PR[GP1:91,1] = PR[GP1:90,1] + 18.194;
   1:  PR[GP1:91,2] = PR[GP1:90,2] + 11.453;
   1:L PR[91] 10mm/sec CNT100;
   1:  PR[GP1:91,1] = PR[GP1:90,1] + 16.157;
   1:  PR[GP1:91,2] = PR[GP1:90,2] + 12.403;
   1:L PR[91] 10mm/sec CNT100;
   1:  PR[GP1:91,1] = PR[GP1:90,1] + 12.851;
   1:  PR[GP1:91,2] = PR[GP1:90,2] + 13.219;
   1:L PR[91] 10mm/sec CNT100;
   1:  PR[GP1:91,1] = PR[GP1:90,1] + 9.521;
   1:  PR[GP1:91,2] = PR[GP1:90,2] + 13.369;
   1:L PR[91] 10mm/sec CNT100;
   1:  PR[GP1:91,1] = PR[GP1:90,1] + 6.108;
   1:  PR[GP1:91,2] = PR[GP1:90,2] + 12.889;
   1:L PR[91] 10mm/sec CNT100;
   1:  PR[GP1:91,1] = PR[GP1:90,1] + 4.989;
   1:  PR[GP1:91,2] = PR[GP1:90,2] + 12.530;
   1:L PR[91] 10mm/sec CNT100;
   1:  PR[GP1:91,1] = PR[GP1:90,1] + 3.048;
   1:  PR[GP1:91,2] = PR[GP1:90,2] + 11.857;
   1:L PR[91] 10mm/sec CNT100;
   1:  PR[GP1:91,1] = PR[GP1:90,1] + 1.753;
   1:  PR[GP1:91,2] = PR[GP1:90,2] + 11.664;
   1:L PR[91] 10mm/sec CNT100;
   1:  PR[GP1:91,1] = PR[GP1:90,1] + -0.697;
   1:  PR[GP1:91,2] = PR[GP1:90,2] + 12.241;
   1:L PR[91] 10mm/sec CNT100;
   1:  PR[GP1:91,1] = PR[GP1:90,1] + -3.443;
   1:  PR[GP1:91,2] = PR[GP1:90,2] + 12.703;
   1:L PR[91] 10mm/sec CNT100;
   1:  PR[GP1:91,1] = PR[GP1:90,1] + -5.012;
   1:  PR[GP1:91,2] = PR[GP1:90,2] + 12.904;
   1:L PR[91] 10mm/sec CNT100;
   1:  PR[GP1:91,1] = PR[GP1:90,1] + -7.309;
   1:  PR[GP1:91,2] = PR[GP1:90,2] + 12.950;
   1:L PR[91] 10mm/sec CNT100;
   1:  PR[GP1:91,1] = PR[GP1:90,1] + -8.564;
   1:  PR[GP1:91,2] = PR[GP1:90,2] + 12.957;
   1:L PR[91] 10mm/sec CNT100;
   1:  PR[GP1:91,1] = PR[GP1:90,1] + -11.248;
   1:  PR[GP1:91,2] = PR[GP1:90,2] + 12.698;
   1:L PR[91] 10mm/sec CNT100;
   1:  PR[GP1:91,1] = PR[GP1:90,1] + -11.480;
   1:  PR[GP1:91,2] = PR[GP1:90,2] + 12.660;
   1:L PR[91] 10mm/sec CNT100;
   1:  PR[GP1:91,1] = PR[GP1:90,1] + -12.466;
   1:  PR[GP1:91,2] = PR[GP1:90,2] + 12.446;
   1:L PR[91] 10mm/sec CNT100;
   1:  PR[GP1:91,1] = PR[GP1:90,1] + -14.278;
   1:  PR[GP1:91,2] = PR[GP1:90,2] + 11.998;
   1:L PR[91] 10mm/sec CNT100;
   1:  PR[GP1:91,1] = PR[GP1:90,1] + -16.083;
   1:  PR[GP1:91,2] = PR[GP1:90,2] + 11.309;
   1:L PR[91] 10mm/sec CNT100;
   1:  PR[GP1:91,1] = PR[GP1:90,1] + -17.401;
   1:  PR[GP1:91,2] = PR[GP1:90,2] + 10.716;
   1:L PR[91] 10mm/sec CNT100;
   1:  PR[GP1:91,1] = PR[GP1:90,1] + -18.604;
   1:  PR[GP1:91,2] = PR[GP1:90,2] + 10.059;
   1:L PR[91] 10mm/sec CNT100;
   1:  PR[GP1:91,1] = PR[GP1:90,1] + -20.478;
   1:  PR[GP1:91,2] = PR[GP1:90,2] + 8.727;
   1:L PR[91] 10mm/sec CNT100;
   1:  PR[GP1:91,1] = PR[GP1:90,1] + -21.133;
   1:  PR[GP1:91,2] = PR[GP1:90,2] + 8.232;
   1:L PR[91] 10mm/sec CNT100;
   1:  PR[GP1:91,1] = PR[GP1:90,1] + -21.536;
   1:  PR[GP1:91,2] = PR[GP1:90,2] + 7.810;
   1:L PR[91] 10mm/sec CNT100;
   1:  PR[GP1:91,1] = PR[GP1:90,1] + -23.361;
   1:  PR[GP1:91,2] = PR[GP1:90,2] + 5.792;
   1:L PR[91] 10mm/sec CNT100;
   1:  PR[GP1:91,1] = PR[GP1:90,1] + -23.529;
   1:  PR[GP1:91,2] = PR[GP1:90,2] + 5.547;
   1:L PR[91] 10mm/sec CNT100;
   1:  PR[GP1:91,1] = PR[GP1:90,1] + -25.024;
   1:  PR[GP1:91,2] = PR[GP1:90,2] + 2.882;
   1:L PR[91] 10mm/sec CNT100;
   1:  PR[GP1:91,1] = PR[GP1:90,1] + -25.078;
   1:  PR[GP1:91,2] = PR[GP1:90,2] + 2.767;
   1:L PR[91] 10mm/sec CNT100;
   1:  PR[GP1:91,1] = PR[GP1:90,1] + -26.012;
   1:  PR[GP1:91,2] = PR[GP1:90,2] + -0.343;
   1:L PR[91] 10mm/sec CNT100;
   1:  PR[GP1:91,1] = PR[GP1:90,1] + -26.018;
   1:  PR[GP1:91,2] = PR[GP1:90,2] + -0.398;
   1:L PR[91] 10mm/sec CNT100;
   1:  PR[GP1:91,1] = PR[GP1:90,1] + -26.068;
   1:  PR[GP1:91,2] = PR[GP1:90,2] + -3.484;
   1:L PR[91] 10mm/sec CNT100;
   1:  PR[GP1:91,1] = PR[GP1:90,1] + -26.055;
   1:  PR[GP1:91,2] = PR[GP1:90,2] + -3.668;
   1:L PR[91] 10mm/sec CNT100;
   1:  PR[GP1:91,1] = PR[GP1:90,1] + -25.455;
   1:  PR[GP1:91,2] = PR[GP1:90,2] + -6.386;
   1:L PR[91] 10mm/sec CNT100;
   1:  PR[GP1:91,1] = PR[GP1:90,1] + -25.288;
   1:  PR[GP1:91,2] = PR[GP1:90,2] + -7.109;
   1:L PR[91] 10mm/sec CNT100;
   1:  PR[GP1:91,1] = PR[GP1:90,1] + -24.949;
   1:  PR[GP1:91,2] = PR[GP1:90,2] + -7.948;
   1:L PR[91] 10mm/sec CNT100;
   1:  PR[GP1:91,1] = PR[GP1:90,1] + -23.999;
   1:  PR[GP1:91,2] = PR[GP1:90,2] + -10.137;
   1:L PR[91] 10mm/sec CNT100;
   1:  PR[GP1:91,1] = PR[GP1:90,1] + -23.203;
   1:  PR[GP1:91,2] = PR[GP1:90,2] + -11.401;
   1:L PR[91] 10mm/sec CNT100;
   1:  PR[GP1:91,1] = PR[GP1:90,1] + -22.293;
   1:  PR[GP1:91,2] = PR[GP1:90,2] + -12.670;
   1:L PR[91] 10mm/sec CNT100;
   1:  PR[GP1:91,1] = PR[GP1:90,1] + -20.754;
   1:  PR[GP1:91,2] = PR[GP1:90,2] + -14.423;
   1:L PR[91] 10mm/sec CNT100;
   1:  PR[GP1:91,1] = PR[GP1:90,1] + -19.738;
   1:  PR[GP1:91,2] = PR[GP1:90,2] + -14.859;
   1:  PR[GP1:91,3] = PR[GP1:90,3] + 40.700;
   1:L PR[91] 10mm/sec CNT100;
   1:  PR[GP1:91,1] = PR[GP1:90,1] + -17.355;
   1:  PR[GP1:91,2] = PR[GP1:90,2] + -16.907;
   1:L PR[91] 10mm/sec CNT100;
   1:  PR[GP1:91,1] = PR[GP1:90,1] + -16.340;
   1:  PR[GP1:91,2] = PR[GP1:90,2] + -17.600;
   1:L PR[91] 10mm/sec CNT100;
   1:  PR[GP1:91,1] = PR[GP1:90,1] + -14.066;
   1:  PR[GP1:91,2] = PR[GP1:90,2] + -19.080;
   1:L PR[91] 10mm/sec CNT100;
   1:  PR[GP1:91,1] = PR[GP1:90,1] + -12.386;
   1:  PR[GP1:91,2] = PR[GP1:90,2] + -19.897;
   1:L PR[91] 10mm/sec CNT100;
   1:  PR[GP1:91,1] = PR[GP1:90,1] + -9.614;
   1:  PR[GP1:91,2] = PR[GP1:90,2] + -21.113;
   1:L PR[91] 10mm/sec CNT100;
   1:  PR[GP1:91,1] = PR[GP1:90,1] + -8.530;
   1:  PR[GP1:91,2] = PR[GP1:90,2] + -21.490;
   1:L PR[91] 10mm/sec CNT100;
   1:  PR[GP1:91,1] = PR[GP1:90,1] + -3.619;
   1:  PR[GP1:91,2] = PR[GP1:90,2] + -22.662;
   1:L PR[91] 10mm/sec CNT100;
   1:  PR[GP1:91,1] = PR[GP1:90,1] + -3.391;
   1:  PR[GP1:91,2] = PR[GP1:90,2] + -22.676;
   1:L PR[91] 10mm/sec CNT100;
   1:  PR[GP1:91,1] = PR[GP1:90,1] + 1.021;
   1:  PR[GP1:91,2] = PR[GP1:90,2] + -23.151;
   1:L PR[91] 10mm/sec CNT100;
   1:  PR[GP1:91,1] = PR[GP1:90,1] + 2.328;
   1:  PR[GP1:91,2] = PR[GP1:90,2] + -23.205;
   1:L PR[91] 10mm/sec CNT100;
   1:  PR[GP1:91,1] = PR[GP1:90,1] + 3.276;
   1:  PR[GP1:91,2] = PR[GP1:90,2] + -23.100;
   1:L PR[91] 10mm/sec CNT100;
   1:  PR[GP1:91,1] = PR[GP1:90,1] + 5.246;
   1:  PR[GP1:91,2] = PR[GP1:90,2] + -22.916;
   1:L PR[91] 10mm/sec CNT100;
   1:  PR[GP1:91,1] = PR[GP1:90,1] + 6.156;
   1:  PR[GP1:91,2] = PR[GP1:90,2] + -22.972;
   1:L PR[91] 10mm/sec CNT100;
   1:  PR[GP1:91,1] = PR[GP1:90,1] + 6.434;
   1:  PR[GP1:91,2] = PR[GP1:90,2] + -23.032;
   1:L PR[91] 10mm/sec CNT100;
   1:  PR[GP1:91,1] = PR[GP1:90,1] + 9.003;
   1:  PR[GP1:91,2] = PR[GP1:90,2] + -23.421;
   1:L PR[91] 10mm/sec CNT100;
   1:  PR[GP1:91,1] = PR[GP1:90,1] + 11.655;
   1:  PR[GP1:91,2] = PR[GP1:90,2] + -23.423;
   1:L PR[91] 10mm/sec CNT100;
   1:  PR[GP1:91,1] = PR[GP1:90,1] + 11.901;
   1:  PR[GP1:91,2] = PR[GP1:90,2] + -23.402;
   1:L PR[91] 10mm/sec CNT100;
   1:  PR[GP1:91,1] = PR[GP1:90,1] + 14.264;
   1:  PR[GP1:91,2] = PR[GP1:90,2] + -23.020;
   1:L PR[91] 10mm/sec CNT100;
   1:  PR[GP1:91,1] = PR[GP1:90,1] + 14.677;
   1:  PR[GP1:91,2] = PR[GP1:90,2] + -22.914;
   1:L PR[91] 10mm/sec CNT100;
   1:  PR[GP1:91,1] = PR[GP1:90,1] + 16.804;
   1:  PR[GP1:91,2] = PR[GP1:90,2] + -22.204;
   1:L PR[91] 10mm/sec CNT100;
   1:  PR[GP1:91,1] = PR[GP1:90,1] + 17.277;
   1:  PR[GP1:91,2] = PR[GP1:90,2] + -21.994;
   1:L PR[91] 10mm/sec CNT100;
   1:  PR[GP1:91,1] = PR[GP1:90,1] + 19.212;
   1:  PR[GP1:91,2] = PR[GP1:90,2] + -20.974;
   1:L PR[91] 10mm/sec CNT100;
   1:  PR[GP1:91,1] = PR[GP1:90,1] + 19.625;
   1:  PR[GP1:91,2] = PR[GP1:90,2] + -20.700;
   1:L PR[91] 10mm/sec CNT100;
   1:  PR[GP1:91,1] = PR[GP1:90,1] + 21.420;
   1:  PR[GP1:91,2] = PR[GP1:90,2] + -19.338;
   1:L PR[91] 10mm/sec CNT100;
   1:  PR[GP1:91,1] = PR[GP1:90,1] + 21.669;
   1:  PR[GP1:91,2] = PR[GP1:90,2] + -19.105;
   1:L PR[91] 10mm/sec CNT100;
   1:  PR[GP1:91,1] = PR[GP1:90,1] + 23.346;
   1:  PR[GP1:91,2] = PR[GP1:90,2] + -17.334;
   1:L PR[91] 10mm/sec CNT100;
   1:  PR[GP1:91,1] = PR[GP1:90,1] + 24.914;
   1:  PR[GP1:91,2] = PR[GP1:90,2] + -15.110;
   1:L PR[91] 10mm/sec CNT100;
   1:  PR[GP1:91,1] = PR[GP1:90,1] + 26.145;
   1:  PR[GP1:91,2] = PR[GP1:90,2] + -12.668;
   1:L PR[91] 10mm/sec CNT100;
   1:  PR[GP1:91,1] = PR[GP1:90,1] + 27.032;
   1:  PR[GP1:91,2] = PR[GP1:90,2] + -9.994;
   1:L PR[91] 10mm/sec CNT100;
   1:  PR[GP1:91,1] = PR[GP1:90,1] + 27.519;
   1:  PR[GP1:91,2] = PR[GP1:90,2] + -7.120;
   1:L PR[91] 10mm/sec CNT100;
   1:  PR[GP1:91,1] = PR[GP1:90,1] + 27.592;
   1:  PR[GP1:91,2] = PR[GP1:90,2] + -4.122;
   1:L PR[91] 10mm/sec CNT100;
   1:  PR[GP1:91,1] = PR[GP1:90,1] + 27.041;
   1:  PR[GP1:91,2] = PR[GP1:90,2] + -0.391;
   1:L PR[91] 10mm/sec CNT100;
   1:  PR[GP1:91,1] = PR[GP1:90,1] + 25.899;
   1:  PR[GP1:91,2] = PR[GP1:90,2] + 3.035;
   1:L PR[91] 10mm/sec CNT100;
   1:  PR[GP1:91,1] = PR[GP1:90,1] + 24.819;
   1:  PR[GP1:91,2] = PR[GP1:90,2] + 4.925;
   1:L PR[91] 10mm/sec CNT100;
   1:  PR[GP1:91,1] = PR[GP1:90,1] + 24.136;
   1:  PR[GP1:91,2] = PR[GP1:90,2] + 6.079;
   1:L PR[91] 10mm/sec CNT100;
   1:  PR[GP1:91,1] = PR[GP1:90,1] + 22.904;
   1:  PR[GP1:91,2] = PR[GP1:90,2] + 7.480;
   1:L PR[91] 10mm/sec CNT100;
   1:  PR[GP1:91,1] = PR[GP1:90,1] + 21.839;
   1:  PR[GP1:91,2] = PR[GP1:90,2] + 8.662;
   1:L PR[91] 10mm/sec CNT100;
   1:  PR[GP1:91,1] = PR[GP1:90,1] + 20.341;
   1:  PR[GP1:91,2] = PR[GP1:90,2] + 9.799;
   1:L PR[91] 10mm/sec CNT100;
   1:  PR[GP1:91,1] = PR[GP1:90,1] + 19.116;
   1:  PR[GP1:91,2] = PR[GP1:90,2] + 10.706;
   1:L PR[91] 10mm/sec CNT100;
   1:  PR[GP1:91,1] = PR[GP1:90,1] + 16.051;
   1:  PR[GP1:91,2] = PR[GP1:90,2] + 12.161;
   1:L PR[91] 10mm/sec CNT100;
   1:  PR[GP1:91,1] = PR[GP1:90,1] + 12.745;
   1:  PR[GP1:91,2] = PR[GP1:90,2] + 12.991;
   1:L PR[91] 10mm/sec CNT100;
   1:  PR[GP1:91,1] = PR[GP1:90,1] + 9.423;
   1:  PR[GP1:91,2] = PR[GP1:90,2] + 13.151;
   1:L PR[91] 10mm/sec CNT100;
   1:  PR[GP1:91,1] = PR[GP1:90,1] + 6.070;
   1:  PR[GP1:91,2] = PR[GP1:90,2] + 12.665;
   1:L PR[91] 10mm/sec CNT100;
   1:  PR[GP1:91,1] = PR[GP1:90,1] + 5.128;
   1:  PR[GP1:91,2] = PR[GP1:90,2] + 12.390;
   1:L PR[91] 10mm/sec CNT100;
   1:  PR[GP1:91,1] = PR[GP1:90,1] + 3.278;
   1:  PR[GP1:91,2] = PR[GP1:90,2] + 11.780;
   1:L PR[91] 10mm/sec CNT100;
   1:  PR[GP1:91,1] = PR[GP1:90,1] + 1.984;
   1:  PR[GP1:91,2] = PR[GP1:90,2] + 11.619;
   1:L PR[91] 10mm/sec CNT100;
   1:  PR[GP1:91,1] = PR[GP1:90,1] + 0.490;
   1:  PR[GP1:91,2] = PR[GP1:90,2] + 11.954;
   1:L PR[91] 10mm/sec CNT100;
   1:  PR[GP1:91,1] = PR[GP1:90,1] + -2.848;
   1:  PR[GP1:91,2] = PR[GP1:90,2] + 12.515;
   1:L PR[91] 10mm/sec CNT100;
   1:  PR[GP1:91,1] = PR[GP1:90,1] + -4.061;
   1:  PR[GP1:91,2] = PR[GP1:90,2] + 12.671;
   1:L PR[91] 10mm/sec CNT100;
   1:  PR[GP1:91,1] = PR[GP1:90,1] + -5.842;
   1:  PR[GP1:91,2] = PR[GP1:90,2] + 12.707;
   1:L PR[91] 10mm/sec CNT100;
   1:  PR[GP1:91,1] = PR[GP1:90,1] + -7.805;
   1:  PR[GP1:91,2] = PR[GP1:90,2] + 12.717;
   1:L PR[91] 10mm/sec CNT100;
   1:  PR[GP1:91,1] = PR[GP1:90,1] + -10.076;
   1:  PR[GP1:91,2] = PR[GP1:90,2] + 12.498;
   1:L PR[91] 10mm/sec CNT100;
   1:  PR[GP1:91,1] = PR[GP1:90,1] + -10.872;
   1:  PR[GP1:91,2] = PR[GP1:90,2] + 12.366;
   1:L PR[91] 10mm/sec CNT100;
   1:  PR[GP1:91,1] = PR[GP1:90,1] + -13.367;
   1:  PR[GP1:91,2] = PR[GP1:90,2] + 11.824;
   1:L PR[91] 10mm/sec CNT100;
   1:  PR[GP1:91,1] = PR[GP1:90,1] + -13.906;
   1:  PR[GP1:91,2] = PR[GP1:90,2] + 11.635;
   1:L PR[91] 10mm/sec CNT100;
   1:  PR[GP1:91,1] = PR[GP1:90,1] + -15.669;
   1:  PR[GP1:91,2] = PR[GP1:90,2] + 10.962;
   1:L PR[91] 10mm/sec CNT100;
   1:  PR[GP1:91,1] = PR[GP1:90,1] + -16.270;
   1:  PR[GP1:91,2] = PR[GP1:90,2] + 10.692;
   1:L PR[91] 10mm/sec CNT100;
   1:  PR[GP1:91,1] = PR[GP1:90,1] + -17.995;
   1:  PR[GP1:91,2] = PR[GP1:90,2] + 9.749;
   1:L PR[91] 10mm/sec CNT100;
   1:  PR[GP1:91,1] = PR[GP1:90,1] + -19.202;
   1:  PR[GP1:91,2] = PR[GP1:90,2] + 8.892;
   1:L PR[91] 10mm/sec CNT100;
   1:  PR[GP1:91,1] = PR[GP1:90,1] + -20.347;
   1:  PR[GP1:91,2] = PR[GP1:90,2] + 8.024;
   1:L PR[91] 10mm/sec CNT100;
   1:  PR[GP1:91,1] = PR[GP1:90,1] + -21.063;
   1:  PR[GP1:91,2] = PR[GP1:90,2] + 7.277;
   1:L PR[91] 10mm/sec CNT100;
   1:  PR[GP1:91,1] = PR[GP1:90,1] + -22.453;
   1:  PR[GP1:91,2] = PR[GP1:90,2] + 5.739;
   1:L PR[91] 10mm/sec CNT100;
   1:  PR[GP1:91,1] = PR[GP1:90,1] + -22.896;
   1:  PR[GP1:91,2] = PR[GP1:90,2] + 5.091;
   1:L PR[91] 10mm/sec CNT100;
   1:  PR[GP1:91,1] = PR[GP1:90,1] + -24.069;
   1:  PR[GP1:91,2] = PR[GP1:90,2] + 3.002;
   1:L PR[91] 10mm/sec CNT100;
   1:  PR[GP1:91,1] = PR[GP1:90,1] + -24.333;
   1:  PR[GP1:91,2] = PR[GP1:90,2] + 2.441;
   1:L PR[91] 10mm/sec CNT100;
   1:  PR[GP1:91,1] = PR[GP1:90,1] + -25.207;
   1:  PR[GP1:91,2] = PR[GP1:90,2] + -0.483;
   1:L PR[91] 10mm/sec CNT100;
   1:  PR[GP1:91,1] = PR[GP1:90,1] + -25.258;
   1:  PR[GP1:91,2] = PR[GP1:90,2] + -0.941;
   1:L PR[91] 10mm/sec CNT100;
   1:  PR[GP1:91,1] = PR[GP1:90,1] + -25.297;
   1:  PR[GP1:91,2] = PR[GP1:90,2] + -3.381;
   1:L PR[91] 10mm/sec CNT100;
   1:  PR[GP1:91,1] = PR[GP1:90,1] + -25.258;
   1:  PR[GP1:91,2] = PR[GP1:90,2] + -3.921;
   1:L PR[91] 10mm/sec CNT100;
   1:  PR[GP1:91,1] = PR[GP1:90,1] + -24.792;
   1:  PR[GP1:91,2] = PR[GP1:90,2] + -6.033;
   1:L PR[91] 10mm/sec CNT100;
   1:  PR[GP1:91,1] = PR[GP1:90,1] + -24.499;
   1:  PR[GP1:91,2] = PR[GP1:90,2] + -7.306;
   1:L PR[91] 10mm/sec CNT100;
   1:  PR[GP1:91,1] = PR[GP1:90,1] + -23.904;
   1:  PR[GP1:91,2] = PR[GP1:90,2] + -8.777;
   1:L PR[91] 10mm/sec CNT100;
   1:  PR[GP1:91,1] = PR[GP1:90,1] + -23.279;
   1:  PR[GP1:91,2] = PR[GP1:90,2] + -10.217;
   1:L PR[91] 10mm/sec CNT100;
   1:  PR[GP1:91,1] = PR[GP1:90,1] + -22.132;
   1:  PR[GP1:91,2] = PR[GP1:90,2] + -12.039;
   1:L PR[91] 10mm/sec CNT100;
   1:  PR[GP1:91,1] = PR[GP1:90,1] + -21.702;
   1:  PR[GP1:91,2] = PR[GP1:90,2] + -12.638;
   1:L PR[91] 10mm/sec CNT100;
   1:  PR[GP1:91,1] = PR[GP1:90,1] + -19.830;
   1:  PR[GP1:91,2] = PR[GP1:90,2] + -14.765;
   1:L PR[91] 10mm/sec CNT100;
   1:  PR[GP1:91,1] = PR[GP1:90,1] + -18.662;
   1:  PR[GP1:91,2] = PR[GP1:90,2] + -15.318;
   1:  PR[GP1:91,3] = PR[GP1:90,3] + 41.800;
   1:L PR[91] 10mm/sec CNT100;
   1:  PR[GP1:91,1] = PR[GP1:90,1] + -16.597;
   1:  PR[GP1:91,2] = PR[GP1:90,2] + -17.093;
   1:L PR[91] 10mm/sec CNT100;
   1:  PR[GP1:91,1] = PR[GP1:90,1] + -14.986;
   1:  PR[GP1:91,2] = PR[GP1:90,2] + -18.191;
   1:L PR[91] 10mm/sec CNT100;
   1:  PR[GP1:91,1] = PR[GP1:90,1] + -13.153;
   1:  PR[GP1:91,2] = PR[GP1:90,2] + -19.384;
   1:L PR[91] 10mm/sec CNT100;
   1:  PR[GP1:91,1] = PR[GP1:90,1] + -11.803;
   1:  PR[GP1:91,2] = PR[GP1:90,2] + -20.041;
   1:L PR[91] 10mm/sec CNT100;
   1:  PR[GP1:91,1] = PR[GP1:90,1] + -8.466;
   1:  PR[GP1:91,2] = PR[GP1:90,2] + -21.505;
   1:L PR[91] 10mm/sec CNT100;
   1:  PR[GP1:91,1] = PR[GP1:90,1] + -7.806;
   1:  PR[GP1:91,2] = PR[GP1:90,2] + -21.734;
   1:L PR[91] 10mm/sec CNT100;
   1:  PR[GP1:91,1] = PR[GP1:90,1] + -4.526;
   1:  PR[GP1:91,2] = PR[GP1:90,2] + -22.518;
   1:L PR[91] 10mm/sec CNT100;
   1:  PR[GP1:91,1] = PR[GP1:90,1] + -2.970;
   1:  PR[GP1:91,2] = PR[GP1:90,2] + -22.982;
   1:L PR[91] 10mm/sec CNT100;
   1:  PR[GP1:91,1] = PR[GP1:90,1] + -2.509;
   1:  PR[GP1:91,2] = PR[GP1:90,2] + -23.090;
   1:L PR[91] 10mm/sec CNT100;
   1:  PR[GP1:91,1] = PR[GP1:90,1] + 1.565;
   1:  PR[GP1:91,2] = PR[GP1:90,2] + -23.529;
   1:L PR[91] 10mm/sec CNT100;
   1:  PR[GP1:91,1] = PR[GP1:90,1] + 3.467;
   1:  PR[GP1:91,2] = PR[GP1:90,2] + -23.608;
   1:L PR[91] 10mm/sec CNT100;
   1:  PR[GP1:91,1] = PR[GP1:90,1] + 4.208;
   1:  PR[GP1:91,2] = PR[GP1:90,2] + -23.519;
   1:L PR[91] 10mm/sec CNT100;
   1:  PR[GP1:91,1] = PR[GP1:90,1] + 5.812;
   1:  PR[GP1:91,2] = PR[GP1:90,2] + -23.364;
   1:L PR[91] 10mm/sec CNT100;
   1:  PR[GP1:91,1] = PR[GP1:90,1] + 6.637;
   1:  PR[GP1:91,2] = PR[GP1:90,2] + -23.413;
   1:L PR[91] 10mm/sec CNT100;
   1:  PR[GP1:91,1] = PR[GP1:90,1] + 8.901;
   1:  PR[GP1:91,2] = PR[GP1:90,2] + -23.764;
   1:L PR[91] 10mm/sec CNT100;
   1:  PR[GP1:91,1] = PR[GP1:90,1] + 9.644;
   1:  PR[GP1:91,2] = PR[GP1:90,2] + -23.821;
   1:L PR[91] 10mm/sec CNT100;
   1:  PR[GP1:91,1] = PR[GP1:90,1] + 11.525;
   1:  PR[GP1:91,2] = PR[GP1:90,2] + -23.819;
   1:L PR[91] 10mm/sec CNT100;
   1:  PR[GP1:91,1] = PR[GP1:90,1] + 12.562;
   1:  PR[GP1:91,2] = PR[GP1:90,2] + -23.730;
   1:L PR[91] 10mm/sec CNT100;
   1:  PR[GP1:91,1] = PR[GP1:90,1] + 14.141;
   1:  PR[GP1:91,2] = PR[GP1:90,2] + -23.474;
   1:L PR[91] 10mm/sec CNT100;
   1:  PR[GP1:91,1] = PR[GP1:90,1] + 15.380;
   1:  PR[GP1:91,2] = PR[GP1:90,2] + -23.156;
   1:L PR[91] 10mm/sec CNT100;
   1:  PR[GP1:91,1] = PR[GP1:90,1] + 16.699;
   1:  PR[GP1:91,2] = PR[GP1:90,2] + -22.716;
   1:L PR[91] 10mm/sec CNT100;
   1:  PR[GP1:91,1] = PR[GP1:90,1] + 18.007;
   1:  PR[GP1:91,2] = PR[GP1:90,2] + -22.135;
   1:L PR[91] 10mm/sec CNT100;
   1:  PR[GP1:91,1] = PR[GP1:90,1] + 19.137;
   1:  PR[GP1:91,2] = PR[GP1:90,2] + -21.540;
   1:L PR[91] 10mm/sec CNT100;
   1:  PR[GP1:91,1] = PR[GP1:90,1] + 20.360;
   1:  PR[GP1:91,2] = PR[GP1:90,2] + -20.729;
   1:L PR[91] 10mm/sec CNT100;
   1:  PR[GP1:91,1] = PR[GP1:90,1] + 21.386;
   1:  PR[GP1:91,2] = PR[GP1:90,2] + -19.951;
   1:L PR[91] 10mm/sec CNT100;
   1:  PR[GP1:91,1] = PR[GP1:90,1] + 22.382;
   1:  PR[GP1:91,2] = PR[GP1:90,2] + -19.017;
   1:L PR[91] 10mm/sec CNT100;
   1:  PR[GP1:91,1] = PR[GP1:90,1] + 23.372;
   1:  PR[GP1:91,2] = PR[GP1:90,2] + -17.971;
   1:L PR[91] 10mm/sec CNT100;
   1:  PR[GP1:91,1] = PR[GP1:90,1] + 24.043;
   1:  PR[GP1:91,2] = PR[GP1:90,2] + -17.090;
   1:L PR[91] 10mm/sec CNT100;
   1:  PR[GP1:91,1] = PR[GP1:90,1] + 25.022;
   1:  PR[GP1:91,2] = PR[GP1:90,2] + -15.645;
   1:L PR[91] 10mm/sec CNT100;
   1:  PR[GP1:91,1] = PR[GP1:90,1] + 25.351;
   1:  PR[GP1:91,2] = PR[GP1:90,2] + -15.025;
   1:L PR[91] 10mm/sec CNT100;
   1:  PR[GP1:91,1] = PR[GP1:90,1] + 26.278;
   1:  PR[GP1:91,2] = PR[GP1:90,2] + -13.053;
   1:L PR[91] 10mm/sec CNT100;
   1:  PR[GP1:91,1] = PR[GP1:90,1] + 26.578;
   1:  PR[GP1:91,2] = PR[GP1:90,2] + -12.080;
   1:L PR[91] 10mm/sec CNT100;
   1:  PR[GP1:91,1] = PR[GP1:90,1] + 27.150;
   1:  PR[GP1:91,2] = PR[GP1:90,2] + -10.358;
   1:L PR[91] 10mm/sec CNT100;
   1:  PR[GP1:91,1] = PR[GP1:90,1] + 27.635;
   1:  PR[GP1:91,2] = PR[GP1:90,2] + -7.562;
   1:L PR[91] 10mm/sec CNT100;
   1:  PR[GP1:91,1] = PR[GP1:90,1] + 27.651;
   1:  PR[GP1:91,2] = PR[GP1:90,2] + -4.616;
   1:L PR[91] 10mm/sec CNT100;
   1:  PR[GP1:91,1] = PR[GP1:90,1] + 27.470;
   1:  PR[GP1:91,2] = PR[GP1:90,2] + -3.468;
   1:L PR[91] 10mm/sec CNT100;
   1:  PR[GP1:91,1] = PR[GP1:90,1] + 27.098;
   1:  PR[GP1:91,2] = PR[GP1:90,2] + -0.837;
   1:L PR[91] 10mm/sec CNT100;
   1:  PR[GP1:91,1] = PR[GP1:90,1] + 25.895;
   1:  PR[GP1:91,2] = PR[GP1:90,2] + 2.650;
   1:L PR[91] 10mm/sec CNT100;
   1:  PR[GP1:91,1] = PR[GP1:90,1] + 24.077;
   1:  PR[GP1:91,2] = PR[GP1:90,2] + 5.754;
   1:L PR[91] 10mm/sec CNT100;
   1:  PR[GP1:91,1] = PR[GP1:90,1] + 21.771;
   1:  PR[GP1:91,2] = PR[GP1:90,2] + 8.369;
   1:L PR[91] 10mm/sec CNT100;
   1:  PR[GP1:91,1] = PR[GP1:90,1] + 19.034;
   1:  PR[GP1:91,2] = PR[GP1:90,2] + 10.440;
   1:L PR[91] 10mm/sec CNT100;
   1:  PR[GP1:91,1] = PR[GP1:90,1] + 15.952;
   1:  PR[GP1:91,2] = PR[GP1:90,2] + 11.917;
   1:L PR[91] 10mm/sec CNT100;
   1:  PR[GP1:91,1] = PR[GP1:90,1] + 12.736;
   1:  PR[GP1:91,2] = PR[GP1:90,2] + 12.738;
   1:L PR[91] 10mm/sec CNT100;
   1:  PR[GP1:91,1] = PR[GP1:90,1] + 9.322;
   1:  PR[GP1:91,2] = PR[GP1:90,2] + 12.933;
   1:L PR[91] 10mm/sec CNT100;
   1:  PR[GP1:91,1] = PR[GP1:90,1] + 6.040;
   1:  PR[GP1:91,2] = PR[GP1:90,2] + 12.442;
   1:L PR[91] 10mm/sec CNT100;
   1:  PR[GP1:91,1] = PR[GP1:90,1] + 4.417;
   1:  PR[GP1:91,2] = PR[GP1:90,2] + 11.967;
   1:L PR[91] 10mm/sec CNT100;
   1:  PR[GP1:91,1] = PR[GP1:90,1] + 3.526;
   1:  PR[GP1:91,2] = PR[GP1:90,2] + 11.684;
   1:L PR[91] 10mm/sec CNT100;
   1:  PR[GP1:91,1] = PR[GP1:90,1] + 2.233;
   1:  PR[GP1:91,2] = PR[GP1:90,2] + 11.538;
   1:L PR[91] 10mm/sec CNT100;
   1:  PR[GP1:91,1] = PR[GP1:90,1] + 1.671;
   1:  PR[GP1:91,2] = PR[GP1:90,2] + 11.668;
   1:L PR[91] 10mm/sec CNT100;
   1:  PR[GP1:91,1] = PR[GP1:90,1] + -2.254;
   1:  PR[GP1:91,2] = PR[GP1:90,2] + 12.328;
   1:L PR[91] 10mm/sec CNT100;
   1:  PR[GP1:91,1] = PR[GP1:90,1] + -3.110;
   1:  PR[GP1:91,2] = PR[GP1:90,2] + 12.438;
   1:L PR[91] 10mm/sec CNT100;
   1:  PR[GP1:91,1] = PR[GP1:90,1] + -4.376;
   1:  PR[GP1:91,2] = PR[GP1:90,2] + 12.464;
   1:L PR[91] 10mm/sec CNT100;
   1:  PR[GP1:91,1] = PR[GP1:90,1] + -7.046;
   1:  PR[GP1:91,2] = PR[GP1:90,2] + 12.477;
   1:L PR[91] 10mm/sec CNT100;
   1:  PR[GP1:91,1] = PR[GP1:90,1] + -8.904;
   1:  PR[GP1:91,2] = PR[GP1:90,2] + 12.298;
   1:L PR[91] 10mm/sec CNT100;
   1:  PR[GP1:91,1] = PR[GP1:90,1] + -10.264;
   1:  PR[GP1:91,2] = PR[GP1:90,2] + 12.072;
   1:L PR[91] 10mm/sec CNT100;
   1:  PR[GP1:91,1] = PR[GP1:90,1] + -12.420;
   1:  PR[GP1:91,2] = PR[GP1:90,2] + 11.604;
   1:L PR[91] 10mm/sec CNT100;
   1:  PR[GP1:91,1] = PR[GP1:90,1] + -15.201;
   1:  PR[GP1:91,2] = PR[GP1:90,2] + 10.626;
   1:L PR[91] 10mm/sec CNT100;
   1:  PR[GP1:91,1] = PR[GP1:90,1] + -17.387;
   1:  PR[GP1:91,2] = PR[GP1:90,2] + 9.439;
   1:L PR[91] 10mm/sec CNT100;
   1:  PR[GP1:91,1] = PR[GP1:90,1] + -17.926;
   1:  PR[GP1:91,2] = PR[GP1:90,2] + 9.056;
   1:L PR[91] 10mm/sec CNT100;
   1:  PR[GP1:91,1] = PR[GP1:90,1] + -19.562;
   1:  PR[GP1:91,2] = PR[GP1:90,2] + 7.817;
   1:L PR[91] 10mm/sec CNT100;
   1:  PR[GP1:91,1] = PR[GP1:90,1] + -20.590;
   1:  PR[GP1:91,2] = PR[GP1:90,2] + 6.744;
   1:L PR[91] 10mm/sec CNT100;
   1:  PR[GP1:91,1] = PR[GP1:90,1] + -21.546;
   1:  PR[GP1:91,2] = PR[GP1:90,2] + 5.686;
   1:L PR[91] 10mm/sec CNT100;
   1:  PR[GP1:91,1] = PR[GP1:90,1] + -22.264;
   1:  PR[GP1:91,2] = PR[GP1:90,2] + 4.636;
   1:L PR[91] 10mm/sec CNT100;
   1:  PR[GP1:91,1] = PR[GP1:90,1] + -23.114;
   1:  PR[GP1:91,2] = PR[GP1:90,2] + 3.121;
   1:L PR[91] 10mm/sec CNT100;
   1:  PR[GP1:91,1] = PR[GP1:90,1] + -23.588;
   1:  PR[GP1:91,2] = PR[GP1:90,2] + 2.114;
   1:L PR[91] 10mm/sec CNT100;
   1:  PR[GP1:91,1] = PR[GP1:90,1] + -24.401;
   1:  PR[GP1:91,2] = PR[GP1:90,2] + -0.623;
   1:L PR[91] 10mm/sec CNT100;
   1:  PR[GP1:91,1] = PR[GP1:90,1] + -24.498;
   1:  PR[GP1:91,2] = PR[GP1:90,2] + -1.484;
   1:L PR[91] 10mm/sec CNT100;
   1:  PR[GP1:91,1] = PR[GP1:90,1] + -24.527;
   1:  PR[GP1:91,2] = PR[GP1:90,2] + -3.277;
   1:L PR[91] 10mm/sec CNT100;
   1:  PR[GP1:91,1] = PR[GP1:90,1] + -24.461;
   1:  PR[GP1:91,2] = PR[GP1:90,2] + -4.174;
   1:L PR[91] 10mm/sec CNT100;
   1:  PR[GP1:91,1] = PR[GP1:90,1] + -24.129;
   1:  PR[GP1:91,2] = PR[GP1:90,2] + -5.681;
   1:L PR[91] 10mm/sec CNT100;
   1:  PR[GP1:91,1] = PR[GP1:90,1] + -23.709;
   1:  PR[GP1:91,2] = PR[GP1:90,2] + -7.503;
   1:L PR[91] 10mm/sec CNT100;
   1:  PR[GP1:91,1] = PR[GP1:90,1] + -22.858;
   1:  PR[GP1:91,2] = PR[GP1:90,2] + -9.606;
   1:L PR[91] 10mm/sec CNT100;
   1:  PR[GP1:91,1] = PR[GP1:90,1] + -22.558;
   1:  PR[GP1:91,2] = PR[GP1:90,2] + -10.297;
   1:L PR[91] 10mm/sec CNT100;
   1:  PR[GP1:91,1] = PR[GP1:90,1] + -21.086;
   1:  PR[GP1:91,2] = PR[GP1:90,2] + -12.634;
   1:L PR[91] 10mm/sec CNT100;
   1:  PR[GP1:91,1] = PR[GP1:90,1] + -19.154;
   1:  PR[GP1:91,2] = PR[GP1:90,2] + -14.814;
   1:L PR[91] 10mm/sec CNT100;
   1:  PR[GP1:91,1] = PR[GP1:90,1] + -17.585;
   1:  PR[GP1:91,2] = PR[GP1:90,2] + -15.776;
   1:  PR[GP1:91,3] = PR[GP1:90,3] + 42.900;
   1:L PR[91] 10mm/sec CNT100;
   1:  PR[GP1:91,1] = PR[GP1:90,1] + -15.838;
   1:  PR[GP1:91,2] = PR[GP1:90,2] + -17.278;
   1:L PR[91] 10mm/sec CNT100;
   1:  PR[GP1:91,1] = PR[GP1:90,1] + -13.631;
   1:  PR[GP1:91,2] = PR[GP1:90,2] + -18.783;
   1:L PR[91] 10mm/sec CNT100;
   1:  PR[GP1:91,1] = PR[GP1:90,1] + -12.240;
   1:  PR[GP1:91,2] = PR[GP1:90,2] + -19.688;
   1:L PR[91] 10mm/sec CNT100;
   1:  PR[GP1:91,1] = PR[GP1:90,1] + -11.220;
   1:  PR[GP1:91,2] = PR[GP1:90,2] + -20.185;
   1:L PR[91] 10mm/sec CNT100;
   1:  PR[GP1:91,1] = PR[GP1:90,1] + -7.318;
   1:  PR[GP1:91,2] = PR[GP1:90,2] + -21.897;
   1:L PR[91] 10mm/sec CNT100;
   1:  PR[GP1:91,1] = PR[GP1:90,1] + -7.083;
   1:  PR[GP1:91,2] = PR[GP1:90,2] + -21.978;
   1:L PR[91] 10mm/sec CNT100;
   1:  PR[GP1:91,1] = PR[GP1:90,1] + -5.761;
   1:  PR[GP1:91,2] = PR[GP1:90,2] + -22.294;
   1:L PR[91] 10mm/sec CNT100;
   1:  PR[GP1:91,1] = PR[GP1:90,1] + -2.440;
   1:  PR[GP1:91,2] = PR[GP1:90,2] + -23.283;
   1:L PR[91] 10mm/sec CNT100;
   1:  PR[GP1:91,1] = PR[GP1:90,1] + -1.390;
   1:  PR[GP1:91,2] = PR[GP1:90,2] + -23.530;
   1:L PR[91] 10mm/sec CNT100;
   1:  PR[GP1:91,1] = PR[GP1:90,1] + 2.110;
   1:  PR[GP1:91,2] = PR[GP1:90,2] + -23.907;
   1:L PR[91] 10mm/sec CNT100;
   1:  PR[GP1:91,1] = PR[GP1:90,1] + 4.611;
   1:  PR[GP1:91,2] = PR[GP1:90,2] + -24.011;
   1:L PR[91] 10mm/sec CNT100;
   1:  PR[GP1:91,1] = PR[GP1:90,1] + 6.402;
   1:  PR[GP1:91,2] = PR[GP1:90,2] + -23.812;
   1:L PR[91] 10mm/sec CNT100;
   1:  PR[GP1:91,1] = PR[GP1:90,1] + 7.164;
   1:  PR[GP1:91,2] = PR[GP1:90,2] + -23.857;
   1:L PR[91] 10mm/sec CNT100;
   1:  PR[GP1:91,1] = PR[GP1:90,1] + 8.773;
   1:  PR[GP1:91,2] = PR[GP1:90,2] + -24.104;
   1:L PR[91] 10mm/sec CNT100;
   1:  PR[GP1:91,1] = PR[GP1:90,1] + 10.252;
   1:  PR[GP1:91,2] = PR[GP1:90,2] + -24.216;
   1:L PR[91] 10mm/sec CNT100;
   1:  PR[GP1:91,1] = PR[GP1:90,1] + 11.395;
   1:  PR[GP1:91,2] = PR[GP1:90,2] + -24.215;
   1:L PR[91] 10mm/sec CNT100;
   1:  PR[GP1:91,1] = PR[GP1:90,1] + 13.223;
   1:  PR[GP1:91,2] = PR[GP1:90,2] + -24.058;
   1:L PR[91] 10mm/sec CNT100;
   1:  PR[GP1:91,1] = PR[GP1:90,1] + 14.019;
   1:  PR[GP1:91,2] = PR[GP1:90,2] + -23.929;
   1:L PR[91] 10mm/sec CNT100;
   1:  PR[GP1:91,1] = PR[GP1:90,1] + 16.084;
   1:  PR[GP1:91,2] = PR[GP1:90,2] + -23.398;
   1:L PR[91] 10mm/sec CNT100;
   1:  PR[GP1:91,1] = PR[GP1:90,1] + 16.594;
   1:  PR[GP1:91,2] = PR[GP1:90,2] + -23.228;
   1:L PR[91] 10mm/sec CNT100;
   1:  PR[GP1:91,1] = PR[GP1:90,1] + 18.738;
   1:  PR[GP1:91,2] = PR[GP1:90,2] + -22.277;
   1:L PR[91] 10mm/sec CNT100;
   1:  PR[GP1:91,1] = PR[GP1:90,1] + 19.061;
   1:  PR[GP1:91,2] = PR[GP1:90,2] + -22.106;
   1:L PR[91] 10mm/sec CNT100;
   1:  PR[GP1:91,1] = PR[GP1:90,1] + 21.095;
   1:  PR[GP1:91,2] = PR[GP1:90,2] + -20.758;
   1:L PR[91] 10mm/sec CNT100;
   1:  PR[GP1:91,1] = PR[GP1:90,1] + 21.351;
   1:  PR[GP1:91,2] = PR[GP1:90,2] + -20.563;
   1:L PR[91] 10mm/sec CNT100;
   1:  PR[GP1:91,1] = PR[GP1:90,1] + 23.095;
   1:  PR[GP1:91,2] = PR[GP1:90,2] + -18.929;
   1:L PR[91] 10mm/sec CNT100;
   1:  PR[GP1:91,1] = PR[GP1:90,1] + 23.391;
   1:  PR[GP1:91,2] = PR[GP1:90,2] + -18.617;
   1:L PR[91] 10mm/sec CNT100;
   1:  PR[GP1:91,1] = PR[GP1:90,1] + 24.704;
   1:  PR[GP1:91,2] = PR[GP1:90,2] + -16.890;
   1:L PR[91] 10mm/sec CNT100;
   1:  PR[GP1:91,1] = PR[GP1:90,1] + 25.100;
   1:  PR[GP1:91,2] = PR[GP1:90,2] + -16.306;
   1:L PR[91] 10mm/sec CNT100;
   1:  PR[GP1:91,1] = PR[GP1:90,1] + 25.936;
   1:  PR[GP1:91,2] = PR[GP1:90,2] + -14.728;
   1:L PR[91] 10mm/sec CNT100;
   1:  PR[GP1:91,1] = PR[GP1:90,1] + 26.420;
   1:  PR[GP1:91,2] = PR[GP1:90,2] + -13.698;
   1:L PR[91] 10mm/sec CNT100;
   1:  PR[GP1:91,1] = PR[GP1:90,1] + 26.831;
   1:  PR[GP1:91,2] = PR[GP1:90,2] + -12.512;
   1:L PR[91] 10mm/sec CNT100;
   1:  PR[GP1:91,1] = PR[GP1:90,1] + 27.315;
   1:  PR[GP1:91,2] = PR[GP1:90,2] + -10.897;
   1:L PR[91] 10mm/sec CNT100;
   1:  PR[GP1:91,1] = PR[GP1:90,1] + 27.425;
   1:  PR[GP1:91,2] = PR[GP1:90,2] + -10.286;
   1:L PR[91] 10mm/sec CNT100;
   1:  PR[GP1:91,1] = PR[GP1:90,1] + 27.752;
   1:  PR[GP1:91,2] = PR[GP1:90,2] + -8.010;
   1:L PR[91] 10mm/sec CNT100;
   1:  PR[GP1:91,1] = PR[GP1:90,1] + 27.767;
   1:  PR[GP1:91,2] = PR[GP1:90,2] + -5.115;
   1:L PR[91] 10mm/sec CNT100;
   1:  PR[GP1:91,1] = PR[GP1:90,1] + 27.171;
   1:  PR[GP1:91,2] = PR[GP1:90,2] + -1.288;
   1:L PR[91] 10mm/sec CNT100;
   1:  PR[GP1:91,1] = PR[GP1:90,1] + 25.973;
   1:  PR[GP1:91,2] = PR[GP1:90,2] + 2.246;
   1:L PR[91] 10mm/sec CNT100;
   1:  PR[GP1:91,1] = PR[GP1:90,1] + 25.130;
   1:  PR[GP1:91,2] = PR[GP1:90,2] + 3.727;
   1:L PR[91] 10mm/sec CNT100;
   1:  PR[GP1:91,1] = PR[GP1:90,1] + 24.147;
   1:  PR[GP1:91,2] = PR[GP1:90,2] + 5.386;
   1:L PR[91] 10mm/sec CNT100;
   1:  PR[GP1:91,1] = PR[GP1:90,1] + 23.467;
   1:  PR[GP1:91,2] = PR[GP1:90,2] + 6.172;
   1:L PR[91] 10mm/sec CNT100;
   1:  PR[GP1:91,1] = PR[GP1:90,1] + 21.800;
   1:  PR[GP1:91,2] = PR[GP1:90,2] + 8.045;
   1:L PR[91] 10mm/sec CNT100;
   1:  PR[GP1:91,1] = PR[GP1:90,1] + 19.045;
   1:  PR[GP1:91,2] = PR[GP1:90,2] + 10.147;
   1:L PR[91] 10mm/sec CNT100;
   1:  PR[GP1:91,1] = PR[GP1:90,1] + 15.989;
   1:  PR[GP1:91,2] = PR[GP1:90,2] + 11.637;
   1:L PR[91] 10mm/sec CNT100;
   1:  PR[GP1:91,1] = PR[GP1:90,1] + 14.662;
   1:  PR[GP1:91,2] = PR[GP1:90,2] + 11.992;
   1:L PR[91] 10mm/sec CNT100;
   1:  PR[GP1:91,1] = PR[GP1:90,1] + 12.731;
   1:  PR[GP1:91,2] = PR[GP1:90,2] + 12.485;
   1:L PR[91] 10mm/sec CNT100;
   1:  PR[GP1:91,1] = PR[GP1:90,1] + 9.346;
   1:  PR[GP1:91,2] = PR[GP1:90,2] + 12.683;
   1:L PR[91] 10mm/sec CNT100;
   1:  PR[GP1:91,1] = PR[GP1:90,1] + 7.800;
   1:  PR[GP1:91,2] = PR[GP1:90,2] + 12.487;
   1:L PR[91] 10mm/sec CNT100;
   1:  PR[GP1:91,1] = PR[GP1:90,1] + 6.009;
   1:  PR[GP1:91,2] = PR[GP1:90,2] + 12.218;
   1:L PR[91] 10mm/sec CNT100;
   1:  PR[GP1:91,1] = PR[GP1:90,1] + 3.780;
   1:  PR[GP1:91,2] = PR[GP1:90,2] + 11.566;
   1:L PR[91] 10mm/sec CNT100;
   1:  PR[GP1:91,1] = PR[GP1:90,1] + 2.506;
   1:  PR[GP1:91,2] = PR[GP1:90,2] + 11.454;
   1:L PR[91] 10mm/sec CNT100;
   1:  PR[GP1:91,1] = PR[GP1:90,1] + -1.659;
   1:  PR[GP1:91,2] = PR[GP1:90,2] + 12.141;
   1:L PR[91] 10mm/sec CNT100;
   1:  PR[GP1:91,1] = PR[GP1:90,1] + -2.155;
   1:  PR[GP1:91,2] = PR[GP1:90,2] + 12.205;
   1:L PR[91] 10mm/sec CNT100;
   1:  PR[GP1:91,1] = PR[GP1:90,1] + -6.288;
   1:  PR[GP1:91,2] = PR[GP1:90,2] + 12.237;
   1:L PR[91] 10mm/sec CNT100;
   1:  PR[GP1:91,1] = PR[GP1:90,1] + -7.732;
   1:  PR[GP1:91,2] = PR[GP1:90,2] + 12.098;
   1:L PR[91] 10mm/sec CNT100;
   1:  PR[GP1:91,1] = PR[GP1:90,1] + -9.656;
   1:  PR[GP1:91,2] = PR[GP1:90,2] + 11.778;
   1:L PR[91] 10mm/sec CNT100;
   1:  PR[GP1:91,1] = PR[GP1:90,1] + -11.471;
   1:  PR[GP1:91,2] = PR[GP1:90,2] + 11.384;
   1:L PR[91] 10mm/sec CNT100;
   1:  PR[GP1:91,1] = PR[GP1:90,1] + -14.424;
   1:  PR[GP1:91,2] = PR[GP1:90,2] + 10.336;
   1:L PR[91] 10mm/sec CNT100;
   1:  PR[GP1:91,1] = PR[GP1:90,1] + -16.718;
   1:  PR[GP1:91,2] = PR[GP1:90,2] + 9.150;
   1:L PR[91] 10mm/sec CNT100;
   1:  PR[GP1:91,1] = PR[GP1:90,1] + -17.062;
   1:  PR[GP1:91,2] = PR[GP1:90,2] + 8.908;
   1:L PR[91] 10mm/sec CNT100;
   1:  PR[GP1:91,1] = PR[GP1:90,1] + -18.777;
   1:  PR[GP1:91,2] = PR[GP1:90,2] + 7.609;
   1:L PR[91] 10mm/sec CNT100;
   1:  PR[GP1:91,1] = PR[GP1:90,1] + -20.117;
   1:  PR[GP1:91,2] = PR[GP1:90,2] + 6.211;
   1:L PR[91] 10mm/sec CNT100;
   1:  PR[GP1:91,1] = PR[GP1:90,1] + -20.638;
   1:  PR[GP1:91,2] = PR[GP1:90,2] + 5.634;
   1:L PR[91] 10mm/sec CNT100;
   1:  PR[GP1:91,1] = PR[GP1:90,1] + -21.632;
   1:  PR[GP1:91,2] = PR[GP1:90,2] + 4.181;
   1:L PR[91] 10mm/sec CNT100;
   1:  PR[GP1:91,1] = PR[GP1:90,1] + -22.159;
   1:  PR[GP1:91,2] = PR[GP1:90,2] + 3.241;
   1:L PR[91] 10mm/sec CNT100;
   1:  PR[GP1:91,1] = PR[GP1:90,1] + -22.843;
   1:  PR[GP1:91,2] = PR[GP1:90,2] + 1.788;
   1:L PR[91] 10mm/sec CNT100;
   1:  PR[GP1:91,1] = PR[GP1:90,1] + -23.596;
   1:  PR[GP1:91,2] = PR[GP1:90,2] + -0.763;
   1:L PR[91] 10mm/sec CNT100;
   1:  PR[GP1:91,1] = PR[GP1:90,1] + -23.737;
   1:  PR[GP1:91,2] = PR[GP1:90,2] + -2.028;
   1:L PR[91] 10mm/sec CNT100;
   1:  PR[GP1:91,1] = PR[GP1:90,1] + -23.756;
   1:  PR[GP1:91,2] = PR[GP1:90,2] + -3.174;
   1:L PR[91] 10mm/sec CNT100;
   1:  PR[GP1:91,1] = PR[GP1:90,1] + -23.665;
   1:  PR[GP1:91,2] = PR[GP1:90,2] + -4.426;
   1:L PR[91] 10mm/sec CNT100;
   1:  PR[GP1:91,1] = PR[GP1:90,1] + -23.466;
   1:  PR[GP1:91,2] = PR[GP1:90,2] + -5.327;
   1:L PR[91] 10mm/sec CNT100;
   1:  PR[GP1:91,1] = PR[GP1:90,1] + -22.919;
   1:  PR[GP1:91,2] = PR[GP1:90,2] + -7.700;
   1:L PR[91] 10mm/sec CNT100;
   1:  PR[GP1:91,1] = PR[GP1:90,1] + -21.832;
   1:  PR[GP1:91,2] = PR[GP1:90,2] + -10.384;
   1:L PR[91] 10mm/sec CNT100;
   1:  PR[GP1:91,1] = PR[GP1:90,1] + -20.187;
   1:  PR[GP1:91,2] = PR[GP1:90,2] + -12.935;
   1:L PR[91] 10mm/sec CNT100;
   1:  PR[GP1:91,1] = PR[GP1:90,1] + -18.477;
   1:  PR[GP1:91,2] = PR[GP1:90,2] + -14.864;
   1:L PR[91] 10mm/sec CNT100;
   1:  PR[GP1:91,1] = PR[GP1:90,1] + -16.509;
   1:  PR[GP1:91,2] = PR[GP1:90,2] + -16.234;
   1:  PR[GP1:91,3] = PR[GP1:90,3] + 44.000;
   1:L PR[91] 10mm/sec CNT100;
   1:  PR[GP1:91,1] = PR[GP1:90,1] + -15.080;
   1:  PR[GP1:91,2] = PR[GP1:90,2] + -17.463;
   1:L PR[91] 10mm/sec CNT100;
   1:  PR[GP1:91,1] = PR[GP1:90,1] + -12.276;
   1:  PR[GP1:91,2] = PR[GP1:90,2] + -19.375;
   1:L PR[91] 10mm/sec CNT100;
   1:  PR[GP1:91,1] = PR[GP1:90,1] + -11.327;
   1:  PR[GP1:91,2] = PR[GP1:90,2] + -19.993;
   1:L PR[91] 10mm/sec CNT100;
   1:  PR[GP1:91,1] = PR[GP1:90,1] + -10.637;
   1:  PR[GP1:91,2] = PR[GP1:90,2] + -20.328;
   1:L PR[91] 10mm/sec CNT100;
   1:  PR[GP1:91,1] = PR[GP1:90,1] + -6.850;
   1:  PR[GP1:91,2] = PR[GP1:90,2] + -21.990;
   1:L PR[91] 10mm/sec CNT100;
   1:  PR[GP1:91,1] = PR[GP1:90,1] + -6.191;
   1:  PR[GP1:91,2] = PR[GP1:90,2] + -22.310;
   1:L PR[91] 10mm/sec CNT100;
   1:  PR[GP1:91,1] = PR[GP1:90,1] + -1.910;
   1:  PR[GP1:91,2] = PR[GP1:90,2] + -23.584;
   1:L PR[91] 10mm/sec CNT100;
   1:  PR[GP1:91,1] = PR[GP1:90,1] + -0.271;
   1:  PR[GP1:91,2] = PR[GP1:90,2] + -23.969;
   1:L PR[91] 10mm/sec CNT100;
   1:  PR[GP1:91,1] = PR[GP1:90,1] + 2.654;
   1:  PR[GP1:91,2] = PR[GP1:90,2] + -24.285;
   1:L PR[91] 10mm/sec CNT100;
   1:  PR[GP1:91,1] = PR[GP1:90,1] + 5.750;
   1:  PR[GP1:91,2] = PR[GP1:90,2] + -24.413;
   1:L PR[91] 10mm/sec CNT100;
   1:  PR[GP1:91,1] = PR[GP1:90,1] + 7.020;
   1:  PR[GP1:91,2] = PR[GP1:90,2] + -24.262;
   1:L PR[91] 10mm/sec CNT100;
   1:  PR[GP1:91,1] = PR[GP1:90,1] + 7.719;
   1:  PR[GP1:91,2] = PR[GP1:90,2] + -24.302;
   1:L PR[91] 10mm/sec CNT100;
   1:  PR[GP1:91,1] = PR[GP1:90,1] + 8.645;
   1:  PR[GP1:91,2] = PR[GP1:90,2] + -24.444;
   1:L PR[91] 10mm/sec CNT100;
   1:  PR[GP1:91,1] = PR[GP1:90,1] + 10.860;
   1:  PR[GP1:91,2] = PR[GP1:90,2] + -24.612;
   1:L PR[91] 10mm/sec CNT100;
   1:  PR[GP1:91,1] = PR[GP1:90,1] + 11.266;
   1:L PR[91] 10mm/sec CNT100;
   1:  PR[GP1:91,1] = PR[GP1:90,1] + 13.858;
   1:  PR[GP1:91,2] = PR[GP1:90,2] + -24.388;
   1:L PR[91] 10mm/sec CNT100;
   1:  PR[GP1:91,1] = PR[GP1:90,1] + 16.518;
   1:  PR[GP1:91,2] = PR[GP1:90,2] + -23.740;
   1:L PR[91] 10mm/sec CNT100;
   1:  PR[GP1:91,1] = PR[GP1:90,1] + 16.717;
   1:  PR[GP1:91,2] = PR[GP1:90,2] + -23.681;
   1:L PR[91] 10mm/sec CNT100;
   1:  PR[GP1:91,1] = PR[GP1:90,1] + 18.940;
   1:  PR[GP1:91,2] = PR[GP1:90,2] + -22.721;
   1:L PR[91] 10mm/sec CNT100;
   1:  PR[GP1:91,1] = PR[GP1:90,1] + 19.336;
   1:  PR[GP1:91,2] = PR[GP1:90,2] + -22.531;
   1:L PR[91] 10mm/sec CNT100;
   1:  PR[GP1:91,1] = PR[GP1:90,1] + 21.207;
   1:  PR[GP1:91,2] = PR[GP1:90,2] + -21.300;
   1:L PR[91] 10mm/sec CNT100;
   1:  PR[GP1:91,1] = PR[GP1:90,1] + 21.657;
   1:  PR[GP1:91,2] = PR[GP1:90,2] + -20.984;
   1:L PR[91] 10mm/sec CNT100;
   1:  PR[GP1:91,1] = PR[GP1:90,1] + 23.283;
   1:  PR[GP1:91,2] = PR[GP1:90,2] + -19.445;
   1:L PR[91] 10mm/sec CNT100;
   1:  PR[GP1:91,1] = PR[GP1:90,1] + 23.645;
   1:  PR[GP1:91,2] = PR[GP1:90,2] + -19.087;
   1:L PR[91] 10mm/sec CNT100;
   1:  PR[GP1:91,1] = PR[GP1:90,1] + 25.274;
   1:  PR[GP1:91,2] = PR[GP1:90,2] + -16.875;
   1:L PR[91] 10mm/sec CNT100;
   1:  PR[GP1:91,1] = PR[GP1:90,1] + 26.124;
   1:  PR[GP1:91,2] = PR[GP1:90,2] + -15.183;
   1:L PR[91] 10mm/sec CNT100;
   1:  PR[GP1:91,1] = PR[GP1:90,1] + 26.563;
   1:  PR[GP1:91,2] = PR[GP1:90,2] + -14.341;
   1:L PR[91] 10mm/sec CNT100;
   1:  PR[GP1:91,1] = PR[GP1:90,1] + 27.325;
   1:  PR[GP1:91,2] = PR[GP1:90,2] + -12.141;
   1:L PR[91] 10mm/sec CNT100;
   1:  PR[GP1:91,1] = PR[GP1:90,1] + 27.509;
   1:  PR[GP1:91,2] = PR[GP1:90,2] + -11.527;
   1:L PR[91] 10mm/sec CNT100;
   1:  PR[GP1:91,1] = PR[GP1:90,1] + 27.809;
   1:  PR[GP1:91,2] = PR[GP1:90,2] + -9.867;
   1:L PR[91] 10mm/sec CNT100;
   1:  PR[GP1:91,1] = PR[GP1:90,1] + 27.990;
   1:  PR[GP1:91,2] = PR[GP1:90,2] + -8.603;
   1:L PR[91] 10mm/sec CNT100;
   1:  PR[GP1:91,1] = PR[GP1:90,1] + 27.958;
   1:  PR[GP1:91,2] = PR[GP1:90,2] + -5.644;
   1:L PR[91] 10mm/sec CNT100;
   1:  PR[GP1:91,1] = PR[GP1:90,1] + 27.355;
   1:  PR[GP1:91,2] = PR[GP1:90,2] + -1.777;
   1:L PR[91] 10mm/sec CNT100;
   1:  PR[GP1:91,1] = PR[GP1:90,1] + 26.078;
   1:  PR[GP1:91,2] = PR[GP1:90,2] + 1.822;
   1:L PR[91] 10mm/sec CNT100;
   1:  PR[GP1:91,1] = PR[GP1:90,1] + 24.231;
   1:  PR[GP1:91,2] = PR[GP1:90,2] + 5.015;
   1:L PR[91] 10mm/sec CNT100;
   1:  PR[GP1:91,1] = PR[GP1:90,1] + 22.751;
   1:  PR[GP1:91,2] = PR[GP1:90,2] + 6.726;
   1:L PR[91] 10mm/sec CNT100;
   1:  PR[GP1:91,1] = PR[GP1:90,1] + 21.876;
   1:  PR[GP1:91,2] = PR[GP1:90,2] + 7.708;
   1:L PR[91] 10mm/sec CNT100;
   1:  PR[GP1:91,1] = PR[GP1:90,1] + 20.417;
   1:  PR[GP1:91,2] = PR[GP1:90,2] + 8.846;
   1:L PR[91] 10mm/sec CNT100;
   1:  PR[GP1:91,1] = PR[GP1:90,1] + 19.108;
   1:  PR[GP1:91,2] = PR[GP1:90,2] + 9.838;
   1:L PR[91] 10mm/sec CNT100;
   1:  PR[GP1:91,1] = PR[GP1:90,1] + 17.468;
   1:  PR[GP1:91,2] = PR[GP1:90,2] + 10.658;
   1:L PR[91] 10mm/sec CNT100;
   1:  PR[GP1:91,1] = PR[GP1:90,1] + 16.032;
   1:  PR[GP1:91,2] = PR[GP1:90,2] + 11.353;
   1:L PR[91] 10mm/sec CNT100;
   1:  PR[GP1:91,1] = PR[GP1:90,1] + 12.722;
   1:  PR[GP1:91,2] = PR[GP1:90,2] + 12.231;
   1:L PR[91] 10mm/sec CNT100;
   1:  PR[GP1:91,1] = PR[GP1:90,1] + 9.386;
   1:  PR[GP1:91,2] = PR[GP1:90,2] + 12.430;
   1:L PR[91] 10mm/sec CNT100;
   1:  PR[GP1:91,1] = PR[GP1:90,1] + 5.972;
   1:  PR[GP1:91,2] = PR[GP1:90,2] + 11.993;
   1:L PR[91] 10mm/sec CNT100;
   1:  PR[GP1:91,1] = PR[GP1:90,1] + 4.057;
   1:  PR[GP1:91,2] = PR[GP1:90,2] + 11.432;
   1:L PR[91] 10mm/sec CNT100;
   1:  PR[GP1:91,1] = PR[GP1:90,1] + 2.785;
   1:  PR[GP1:91,2] = PR[GP1:90,2] + 11.336;
   1:L PR[91] 10mm/sec CNT100;
   1:  PR[GP1:91,1] = PR[GP1:90,1] + -1.214;
   1:  PR[GP1:91,2] = PR[GP1:90,2] + 11.972;
   1:L PR[91] 10mm/sec CNT100;
   1:  PR[GP1:91,1] = PR[GP1:90,1] + -5.528;
   1:  PR[GP1:91,2] = PR[GP1:90,2] + 11.998;
   1:L PR[91] 10mm/sec CNT100;
   1:  PR[GP1:91,1] = PR[GP1:90,1] + -6.560;
   1:  PR[GP1:91,2] = PR[GP1:90,2] + 11.898;
   1:L PR[91] 10mm/sec CNT100;
   1:  PR[GP1:91,1] = PR[GP1:90,1] + -9.047;
   1:  PR[GP1:91,2] = PR[GP1:90,2] + 11.484;
   1:L PR[91] 10mm/sec CNT100;
   1:  PR[GP1:91,1] = PR[GP1:90,1] + -10.525;
   1:  PR[GP1:91,2] = PR[GP1:90,2] + 11.163;
   1:L PR[91] 10mm/sec CNT100;
   1:  PR[GP1:91,1] = PR[GP1:90,1] + -12.428;
   1:  PR[GP1:91,2] = PR[GP1:90,2] + 10.494;
   1:L PR[91] 10mm/sec CNT100;
   1:  PR[GP1:91,1] = PR[GP1:90,1] + -13.638;
   1:  PR[GP1:91,2] = PR[GP1:90,2] + 10.050;
   1:L PR[91] 10mm/sec CNT100;
   1:  PR[GP1:91,1] = PR[GP1:90,1] + -15.618;
   1:  PR[GP1:91,2] = PR[GP1:90,2] + 9.027;
   1:L PR[91] 10mm/sec CNT100;
   1:  PR[GP1:91,1] = PR[GP1:90,1] + -16.083;
   1:  PR[GP1:91,2] = PR[GP1:90,2] + 8.736;
   1:L PR[91] 10mm/sec CNT100;
   1:  PR[GP1:91,1] = PR[GP1:90,1] + -17.956;
   1:  PR[GP1:91,2] = PR[GP1:90,2] + 7.391;
   1:L PR[91] 10mm/sec CNT100;
   1:  PR[GP1:91,1] = PR[GP1:90,1] + -18.922;
   1:  PR[GP1:91,2] = PR[GP1:90,2] + 6.431;
   1:L PR[91] 10mm/sec CNT100;
   1:  PR[GP1:91,1] = PR[GP1:90,1] + -19.735;
   1:  PR[GP1:91,2] = PR[GP1:90,2] + 5.575;
   1:L PR[91] 10mm/sec CNT100;
   1:  PR[GP1:91,1] = PR[GP1:90,1] + -21.000;
   1:  PR[GP1:91,2] = PR[GP1:90,2] + 3.726;
   1:L PR[91] 10mm/sec CNT100;
   1:  PR[GP1:91,1] = PR[GP1:90,1] + -21.205;
   1:  PR[GP1:91,2] = PR[GP1:90,2] + 3.361;
   1:L PR[91] 10mm/sec CNT100;
   1:  PR[GP1:91,1] = PR[GP1:90,1] + -22.098;
   1:  PR[GP1:91,2] = PR[GP1:90,2] + 1.461;
   1:L PR[91] 10mm/sec CNT100;
   1:  PR[GP1:91,1] = PR[GP1:90,1] + -22.790;
   1:  PR[GP1:91,2] = PR[GP1:90,2] + -0.903;
   1:L PR[91] 10mm/sec CNT100;
   1:  PR[GP1:91,1] = PR[GP1:90,1] + -22.977;
   1:  PR[GP1:91,2] = PR[GP1:90,2] + -2.571;
   1:L PR[91] 10mm/sec CNT100;
   1:  PR[GP1:91,1] = PR[GP1:90,1] + -22.985;
   1:  PR[GP1:91,2] = PR[GP1:90,2] + -3.070;
   1:L PR[91] 10mm/sec CNT100;
   1:  PR[GP1:91,1] = PR[GP1:90,1] + -22.868;
   1:  PR[GP1:91,2] = PR[GP1:90,2] + -4.679;
   1:L PR[91] 10mm/sec CNT100;
   1:  PR[GP1:91,1] = PR[GP1:90,1] + -22.802;
   1:  PR[GP1:91,2] = PR[GP1:90,2] + -4.975;
   1:L PR[91] 10mm/sec CNT100;
   1:  PR[GP1:91,1] = PR[GP1:90,1] + -22.286;
   1:  PR[GP1:91,2] = PR[GP1:90,2] + -7.220;
   1:L PR[91] 10mm/sec CNT100;
   1:  PR[GP1:91,1] = PR[GP1:90,1] + -22.107;
   1:  PR[GP1:91,2] = PR[GP1:90,2] + -7.929;
   1:L PR[91] 10mm/sec CNT100;
   1:  PR[GP1:91,1] = PR[GP1:90,1] + -21.015;
   1:  PR[GP1:91,2] = PR[GP1:90,2] + -10.528;
   1:L PR[91] 10mm/sec CNT100;
   1:  PR[GP1:91,1] = PR[GP1:90,1] + -20.740;
   1:  PR[GP1:91,2] = PR[GP1:90,2] + -10.984;
   1:L PR[91] 10mm/sec CNT100;
   1:  PR[GP1:91,1] = PR[GP1:90,1] + -19.285;
   1:  PR[GP1:91,2] = PR[GP1:90,2] + -13.240;
   1:L PR[91] 10mm/sec CNT100;
   1:  PR[GP1:91,1] = PR[GP1:90,1] + -17.801;
   1:  PR[GP1:91,2] = PR[GP1:90,2] + -14.914;
   1:L PR[91] 10mm/sec CNT100;
   1:  PR[GP1:91,1] = PR[GP1:90,1] + -15.433;
   1:  PR[GP1:91,2] = PR[GP1:90,2] + -16.693;
   1:  PR[GP1:91,3] = PR[GP1:90,3] + 45.100;
   1:L PR[91] 10mm/sec CNT100;
   1:  PR[GP1:91,1] = PR[GP1:90,1] + -14.322;
   1:  PR[GP1:91,2] = PR[GP1:90,2] + -17.648;
   1:L PR[91] 10mm/sec CNT100;
   1:  PR[GP1:91,1] = PR[GP1:90,1] + -10.921;
   1:  PR[GP1:91,2] = PR[GP1:90,2] + -19.967;
   1:L PR[91] 10mm/sec CNT100;
   1:  PR[GP1:91,1] = PR[GP1:90,1] + -10.414;
   1:  PR[GP1:91,2] = PR[GP1:90,2] + -20.297;
   1:L PR[91] 10mm/sec CNT100;
   1:  PR[GP1:91,1] = PR[GP1:90,1] + -10.054;
   1:  PR[GP1:91,2] = PR[GP1:90,2] + -20.472;
   1:L PR[91] 10mm/sec CNT100;
   1:  PR[GP1:91,1] = PR[GP1:90,1] + -7.954;
   1:  PR[GP1:91,2] = PR[GP1:90,2] + -21.394;
   1:L PR[91] 10mm/sec CNT100;
   1:  PR[GP1:91,1] = PR[GP1:90,1] + -5.789;
   1:  PR[GP1:91,2] = PR[GP1:90,2] + -22.481;
   1:L PR[91] 10mm/sec CNT100;
   1:  PR[GP1:91,1] = PR[GP1:90,1] + -5.121;
   1:  PR[GP1:91,2] = PR[GP1:90,2] + -22.772;
   1:L PR[91] 10mm/sec CNT100;
   1:  PR[GP1:91,1] = PR[GP1:90,1] + -1.380;
   1:  PR[GP1:91,2] = PR[GP1:90,2] + -23.886;
   1:L PR[91] 10mm/sec CNT100;
   1:  PR[GP1:91,1] = PR[GP1:90,1] + 0.848;
   1:  PR[GP1:91,2] = PR[GP1:90,2] + -24.409;
   1:L PR[91] 10mm/sec CNT100;
   1:  PR[GP1:91,1] = PR[GP1:90,1] + 3.199;
   1:  PR[GP1:91,2] = PR[GP1:90,2] + -24.662;
   1:L PR[91] 10mm/sec CNT100;
   1:  PR[GP1:91,1] = PR[GP1:90,1] + 6.889;
   1:  PR[GP1:91,2] = PR[GP1:90,2] + -24.816;
   1:L PR[91] 10mm/sec CNT100;
   1:  PR[GP1:91,1] = PR[GP1:90,1] + 7.670;
   1:  PR[GP1:91,2] = PR[GP1:90,2] + -24.715;
   1:L PR[91] 10mm/sec CNT100;
   1:  PR[GP1:91,1] = PR[GP1:90,1] + 8.305;
   1:  PR[GP1:91,2] = PR[GP1:90,2] + -24.751;
   1:L PR[91] 10mm/sec CNT100;
   1:  PR[GP1:91,1] = PR[GP1:90,1] + 8.519;
   1:  PR[GP1:91,2] = PR[GP1:90,2] + -24.784;
   1:L PR[91] 10mm/sec CNT100;
   1:  PR[GP1:91,1] = PR[GP1:90,1] + 11.196;
   1:  PR[GP1:91,2] = PR[GP1:90,2] + -25.006;
   1:L PR[91] 10mm/sec CNT100;
   1:  PR[GP1:91,1] = PR[GP1:90,1] + 11.452;
   1:  PR[GP1:91,2] = PR[GP1:90,2] + -25.014;
   1:L PR[91] 10mm/sec CNT100;
   1:  PR[GP1:91,1] = PR[GP1:90,1] + 13.790;
   1:  PR[GP1:91,2] = PR[GP1:90,2] + -24.846;
   1:L PR[91] 10mm/sec CNT100;
   1:  PR[GP1:91,1] = PR[GP1:90,1] + 14.483;
   1:  PR[GP1:91,2] = PR[GP1:90,2] + -24.757;
   1:L PR[91] 10mm/sec CNT100;
   1:  PR[GP1:91,1] = PR[GP1:90,1] + 16.285;
   1:  PR[GP1:91,2] = PR[GP1:90,2] + -24.320;
   1:L PR[91] 10mm/sec CNT100;
   1:  PR[GP1:91,1] = PR[GP1:90,1] + 17.315;
   1:  PR[GP1:91,2] = PR[GP1:90,2] + -24.018;
   1:L PR[91] 10mm/sec CNT100;
   1:  PR[GP1:91,1] = PR[GP1:90,1] + 18.663;
   1:  PR[GP1:91,2] = PR[GP1:90,2] + -23.436;
   1:L PR[91] 10mm/sec CNT100;
   1:  PR[GP1:91,1] = PR[GP1:90,1] + 19.891;
   1:  PR[GP1:91,2] = PR[GP1:90,2] + -22.848;
   1:L PR[91] 10mm/sec CNT100;
   1:  PR[GP1:91,1] = PR[GP1:90,1] + 20.901;
   1:  PR[GP1:91,2] = PR[GP1:90,2] + -22.183;
   1:L PR[91] 10mm/sec CNT100;
   1:  PR[GP1:91,1] = PR[GP1:90,1] + 22.167;
   1:  PR[GP1:91,2] = PR[GP1:90,2] + -21.294;
   1:L PR[91] 10mm/sec CNT100;
   1:  PR[GP1:91,1] = PR[GP1:90,1] + 22.971;
   1:  PR[GP1:91,2] = PR[GP1:90,2] + -20.533;
   1:L PR[91] 10mm/sec CNT100;
   1:  PR[GP1:91,1] = PR[GP1:90,1] + 24.111;
   1:  PR[GP1:91,2] = PR[GP1:90,2] + -19.407;
   1:L PR[91] 10mm/sec CNT100;
   1:  PR[GP1:91,1] = PR[GP1:90,1] + 25.703;
   1:  PR[GP1:91,2] = PR[GP1:90,2] + -17.216;
   1:L PR[91] 10mm/sec CNT100;
   1:  PR[GP1:91,1] = PR[GP1:90,1] + 26.417;
   1:  PR[GP1:91,2] = PR[GP1:90,2] + -15.793;
   1:L PR[91] 10mm/sec CNT100;
   1:  PR[GP1:91,1] = PR[GP1:90,1] + 26.925;
   1:  PR[GP1:91,2] = PR[GP1:90,2] + -14.768;
   1:L PR[91] 10mm/sec CNT100;
   1:  PR[GP1:91,1] = PR[GP1:90,1] + 27.766;
   1:  PR[GP1:91,2] = PR[GP1:90,2] + -12.093;
   1:L PR[91] 10mm/sec CNT100;
   1:  PR[GP1:91,1] = PR[GP1:90,1] + 27.983;
   1:  PR[GP1:91,2] = PR[GP1:90,2] + -10.610;
   1:L PR[91] 10mm/sec CNT100;
   1:  PR[GP1:91,1] = PR[GP1:90,1] + 28.229;
   1:  PR[GP1:91,2] = PR[GP1:90,2] + -9.183;
   1:L PR[91] 10mm/sec CNT100;
   1:  PR[GP1:91,1] = PR[GP1:90,1] + 28.196;
   1:  PR[GP1:91,2] = PR[GP1:90,2] + -6.181;
   1:L PR[91] 10mm/sec CNT100;
   1:  PR[GP1:91,1] = PR[GP1:90,1] + 27.539;
   1:  PR[GP1:91,2] = PR[GP1:90,2] + -2.262;
   1:L PR[91] 10mm/sec CNT100;
   1:  PR[GP1:91,1] = PR[GP1:90,1] + 26.285;
   1:  PR[GP1:91,2] = PR[GP1:90,2] + 1.374;
   1:L PR[91] 10mm/sec CNT100;
   1:  PR[GP1:91,1] = PR[GP1:90,1] + 25.642;
   1:  PR[GP1:91,2] = PR[GP1:90,2] + 2.500;
   1:L PR[91] 10mm/sec CNT100;
   1:  PR[GP1:91,1] = PR[GP1:90,1] + 24.374;
   1:  PR[GP1:91,2] = PR[GP1:90,2] + 4.618;
   1:L PR[91] 10mm/sec CNT100;
   1:  PR[GP1:91,1] = PR[GP1:90,1] + 21.954;
   1:  PR[GP1:91,2] = PR[GP1:90,2] + 7.369;
   1:L PR[91] 10mm/sec CNT100;
   1:  PR[GP1:91,1] = PR[GP1:90,1] + 19.171;
   1:  PR[GP1:91,2] = PR[GP1:90,2] + 9.529;
   1:L PR[91] 10mm/sec CNT100;
   1:  PR[GP1:91,1] = PR[GP1:90,1] + 16.069;
   1:  PR[GP1:91,2] = PR[GP1:90,2] + 11.072;
   1:L PR[91] 10mm/sec CNT100;
   1:  PR[GP1:91,1] = PR[GP1:90,1] + 12.767;
   1:  PR[GP1:91,2] = PR[GP1:90,2] + 11.963;
   1:L PR[91] 10mm/sec CNT100;
   1:  PR[GP1:91,1] = PR[GP1:90,1] + 11.937;
   1:  PR[GP1:91,2] = PR[GP1:90,2] + 12.026;
   1:L PR[91] 10mm/sec CNT100;
   1:  PR[GP1:91,1] = PR[GP1:90,1] + 9.426;
   1:  PR[GP1:91,2] = PR[GP1:90,2] + 12.178;
   1:L PR[91] 10mm/sec CNT100;
   1:  PR[GP1:91,1] = PR[GP1:90,1] + 6.036;
   1:  PR[GP1:91,2] = PR[GP1:90,2] + 11.738;
   1:L PR[91] 10mm/sec CNT100;
   1:  PR[GP1:91,1] = PR[GP1:90,1] + 5.422;
   1:  PR[GP1:91,2] = PR[GP1:90,2] + 11.587;
   1:L PR[91] 10mm/sec CNT100;
   1:  PR[GP1:91,1] = PR[GP1:90,1] + 4.341;
   1:  PR[GP1:91,2] = PR[GP1:90,2] + 11.280;
   1:L PR[91] 10mm/sec CNT100;
   1:  PR[GP1:91,1] = PR[GP1:90,1] + 3.077;
   1:  PR[GP1:91,2] = PR[GP1:90,2] + 11.211;
   1:L PR[91] 10mm/sec CNT100;
   1:  PR[GP1:91,1] = PR[GP1:90,1] + 0.369;
   1:  PR[GP1:91,2] = PR[GP1:90,2] + 11.631;
   1:L PR[91] 10mm/sec CNT100;
   1:  PR[GP1:91,1] = PR[GP1:90,1] + -0.290;
   1:  PR[GP1:91,2] = PR[GP1:90,2] + 11.717;
   1:L PR[91] 10mm/sec CNT100;
   1:  PR[GP1:91,1] = PR[GP1:90,1] + -1.310;
   1:  PR[GP1:91,2] = PR[GP1:90,2] + 11.741;
   1:L PR[91] 10mm/sec CNT100;
   1:  PR[GP1:91,1] = PR[GP1:90,1] + -4.769;
   1:  PR[GP1:91,2] = PR[GP1:90,2] + 11.758;
   1:L PR[91] 10mm/sec CNT100;
   1:  PR[GP1:91,1] = PR[GP1:90,1] + -5.387;
   1:  PR[GP1:91,2] = PR[GP1:90,2] + 11.698;
   1:L PR[91] 10mm/sec CNT100;
   1:  PR[GP1:91,1] = PR[GP1:90,1] + -8.439;
   1:  PR[GP1:91,2] = PR[GP1:90,2] + 11.190;
   1:L PR[91] 10mm/sec CNT100;
   1:  PR[GP1:91,1] = PR[GP1:90,1] + -9.577;
   1:  PR[GP1:91,2] = PR[GP1:90,2] + 10.943;
   1:L PR[91] 10mm/sec CNT100;
   1:  PR[GP1:91,1] = PR[GP1:90,1] + -11.050;
   1:  PR[GP1:91,2] = PR[GP1:90,2] + 10.425;
   1:L PR[91] 10mm/sec CNT100;
   1:  PR[GP1:91,1] = PR[GP1:90,1] + -12.856;
   1:  PR[GP1:91,2] = PR[GP1:90,2] + 9.762;
   1:L PR[91] 10mm/sec CNT100;
   1:  PR[GP1:91,1] = PR[GP1:90,1] + -14.502;
   1:  PR[GP1:91,2] = PR[GP1:90,2] + 8.911;
   1:L PR[91] 10mm/sec CNT100;
   1:  PR[GP1:91,1] = PR[GP1:90,1] + -15.415;
   1:  PR[GP1:91,2] = PR[GP1:90,2] + 8.340;
   1:L PR[91] 10mm/sec CNT100;
   1:  PR[GP1:91,1] = PR[GP1:90,1] + -17.024;
   1:  PR[GP1:91,2] = PR[GP1:90,2] + 7.185;
   1:L PR[91] 10mm/sec CNT100;
   1:  PR[GP1:91,1] = PR[GP1:90,1] + -18.901;
   1:  PR[GP1:91,2] = PR[GP1:90,2] + 5.312;
   1:L PR[91] 10mm/sec CNT100;
   1:  PR[GP1:91,1] = PR[GP1:90,1] + -20.250;
   1:  PR[GP1:91,2] = PR[GP1:90,2] + 3.398;
   1:L PR[91] 10mm/sec CNT100;
   1:  PR[GP1:91,1] = PR[GP1:90,1] + -21.346;
   1:  PR[GP1:91,2] = PR[GP1:90,2] + 1.137;
   1:L PR[91] 10mm/sec CNT100;
   1:  PR[GP1:91,1] = PR[GP1:90,1] + -21.984;
   1:  PR[GP1:91,2] = PR[GP1:90,2] + -1.041;
   1:L PR[91] 10mm/sec CNT100;
   1:  PR[GP1:91,1] = PR[GP1:90,1] + -22.195;
   1:  PR[GP1:91,2] = PR[GP1:90,2] + -3.015;
   1:L PR[91] 10mm/sec CNT100;
   1:  PR[GP1:91,1] = PR[GP1:90,1] + -22.033;
   1:  PR[GP1:91,2] = PR[GP1:90,2] + -4.806;
   1:L PR[91] 10mm/sec CNT100;
   1:  PR[GP1:91,1] = PR[GP1:90,1] + -22.028;
   1:  PR[GP1:91,2] = PR[GP1:90,2] + -4.967;
   1:L PR[91] 10mm/sec CNT100;
   1:  PR[GP1:91,1] = PR[GP1:90,1] + -21.317;
   1:  PR[GP1:91,2] = PR[GP1:90,2] + -7.877;
   1:L PR[91] 10mm/sec CNT100;
   1:  PR[GP1:91,1] = PR[GP1:90,1] + -21.163;
   1:  PR[GP1:91,2] = PR[GP1:90,2] + -8.370;
   1:L PR[91] 10mm/sec CNT100;
   1:  PR[GP1:91,1] = PR[GP1:90,1] + -20.197;
   1:  PR[GP1:91,2] = PR[GP1:90,2] + -10.669;
   1:L PR[91] 10mm/sec CNT100;
   1:  PR[GP1:91,1] = PR[GP1:90,1] + -19.618;
   1:  PR[GP1:91,2] = PR[GP1:90,2] + -11.628;
   1:L PR[91] 10mm/sec CNT100;
   1:  PR[GP1:91,1] = PR[GP1:90,1] + -18.383;
   1:  PR[GP1:91,2] = PR[GP1:90,2] + -13.544;
   1:L PR[91] 10mm/sec CNT100;
   1:  PR[GP1:91,1] = PR[GP1:90,1] + -17.124;
   1:  PR[GP1:91,2] = PR[GP1:90,2] + -14.964;
   1:L PR[91] 10mm/sec CNT100;
   1:  PR[GP1:91,1] = PR[GP1:90,1] + -14.356;
   1:  PR[GP1:91,2] = PR[GP1:90,2] + -17.151;
   1:  PR[GP1:91,3] = PR[GP1:90,3] + 46.200;
   1:L PR[91] 10mm/sec CNT100;
   1:  PR[GP1:91,1] = PR[GP1:90,1] + -13.563;
   1:  PR[GP1:91,2] = PR[GP1:90,2] + -17.833;
   1:L PR[91] 10mm/sec CNT100;
   1:  PR[GP1:91,1] = PR[GP1:90,1] + -9.504;
   1:  PR[GP1:91,2] = PR[GP1:90,2] + -20.598;
   1:L PR[91] 10mm/sec CNT100;
   1:  PR[GP1:91,1] = PR[GP1:90,1] + -9.061;
   1:  PR[GP1:91,2] = PR[GP1:90,2] + -20.796;
   1:L PR[91] 10mm/sec CNT100;
   1:  PR[GP1:91,1] = PR[GP1:90,1] + -5.252;
   1:  PR[GP1:91,2] = PR[GP1:90,2] + -22.709;
   1:L PR[91] 10mm/sec CNT100;
   1:  PR[GP1:91,1] = PR[GP1:90,1] + -4.038;
   1:  PR[GP1:91,2] = PR[GP1:90,2] + -23.238;
   1:L PR[91] 10mm/sec CNT100;
   1:  PR[GP1:91,1] = PR[GP1:90,1] + -0.850;
   1:  PR[GP1:91,2] = PR[GP1:90,2] + -24.187;
   1:L PR[91] 10mm/sec CNT100;
   1:  PR[GP1:91,1] = PR[GP1:90,1] + 1.967;
   1:  PR[GP1:91,2] = PR[GP1:90,2] + -24.849;
   1:L PR[91] 10mm/sec CNT100;
   1:  PR[GP1:91,1] = PR[GP1:90,1] + 3.743;
   1:  PR[GP1:91,2] = PR[GP1:90,2] + -25.040;
   1:L PR[91] 10mm/sec CNT100;
   1:  PR[GP1:91,1] = PR[GP1:90,1] + 8.027;
   1:  PR[GP1:91,2] = PR[GP1:90,2] + -25.218;
   1:L PR[91] 10mm/sec CNT100;
   1:  PR[GP1:91,1] = PR[GP1:90,1] + 8.351;
   1:  PR[GP1:91,2] = PR[GP1:90,2] + -25.173;
   1:L PR[91] 10mm/sec CNT100;
   1:  PR[GP1:91,1] = PR[GP1:90,1] + 8.909;
   1:  PR[GP1:91,2] = PR[GP1:90,2] + -25.204;
   1:L PR[91] 10mm/sec CNT100;
   1:  PR[GP1:91,1] = PR[GP1:90,1] + 11.082;
   1:  PR[GP1:91,2] = PR[GP1:90,2] + -25.398;
   1:L PR[91] 10mm/sec CNT100;
   1:  PR[GP1:91,1] = PR[GP1:90,1] + 12.119;
   1:  PR[GP1:91,2] = PR[GP1:90,2] + -25.427;
   1:L PR[91] 10mm/sec CNT100;
   1:  PR[GP1:91,1] = PR[GP1:90,1] + 13.610;
   1:  PR[GP1:91,2] = PR[GP1:90,2] + -25.320;
   1:L PR[91] 10mm/sec CNT100;
   1:  PR[GP1:91,1] = PR[GP1:90,1] + 15.119;
   1:  PR[GP1:91,2] = PR[GP1:90,2] + -25.127;
   1:L PR[91] 10mm/sec CNT100;
   1:  PR[GP1:91,1] = PR[GP1:90,1] + 16.052;
   1:  PR[GP1:91,2] = PR[GP1:90,2] + -24.901;
   1:L PR[91] 10mm/sec CNT100;
   1:  PR[GP1:91,1] = PR[GP1:90,1] + 17.913;
   1:  PR[GP1:91,2] = PR[GP1:90,2] + -24.356;
   1:L PR[91] 10mm/sec CNT100;
   1:  PR[GP1:91,1] = PR[GP1:90,1] + 18.386;
   1:  PR[GP1:91,2] = PR[GP1:90,2] + -24.151;
   1:L PR[91] 10mm/sec CNT100;
   1:  PR[GP1:91,1] = PR[GP1:90,1] + 20.446;
   1:  PR[GP1:91,2] = PR[GP1:90,2] + -23.165;
   1:L PR[91] 10mm/sec CNT100;
   1:  PR[GP1:91,1] = PR[GP1:90,1] + 20.595;
   1:  PR[GP1:91,2] = PR[GP1:90,2] + -23.067;
   1:L PR[91] 10mm/sec CNT100;
   1:  PR[GP1:91,1] = PR[GP1:90,1] + 22.672;
   1:  PR[GP1:91,2] = PR[GP1:90,2] + -21.608;
   1:L PR[91] 10mm/sec CNT100;
   1:  PR[GP1:91,1] = PR[GP1:90,1] + 24.576;
   1:  PR[GP1:91,2] = PR[GP1:90,2] + -19.726;
   1:L PR[91] 10mm/sec CNT100;
   1:  PR[GP1:91,1] = PR[GP1:90,1] + 26.131;
   1:  PR[GP1:91,2] = PR[GP1:90,2] + -17.559;
   1:L PR[91] 10mm/sec CNT100;
   1:  PR[GP1:91,1] = PR[GP1:90,1] + 27.328;
   1:  PR[GP1:91,2] = PR[GP1:90,2] + -15.143;
   1:L PR[91] 10mm/sec CNT100;
   1:  PR[GP1:91,1] = PR[GP1:90,1] + 28.156;
   1:  PR[GP1:91,2] = PR[GP1:90,2] + -12.514;
   1:L PR[91] 10mm/sec CNT100;
   1:  PR[GP1:91,1] = PR[GP1:90,1] + 28.571;
   1:  PR[GP1:91,2] = PR[GP1:90,2] + -9.704;
   1:L PR[91] 10mm/sec CNT100;
   1:  PR[GP1:91,1] = PR[GP1:90,1] + 28.503;
   1:  PR[GP1:91,2] = PR[GP1:90,2] + -6.722;
   1:L PR[91] 10mm/sec CNT100;
   1:  PR[GP1:91,1] = PR[GP1:90,1] + 27.846;
   1:  PR[GP1:91,2] = PR[GP1:90,2] + -2.780;
   1:L PR[91] 10mm/sec CNT100;
   1:  PR[GP1:91,1] = PR[GP1:90,1] + 26.700;
   1:  PR[GP1:91,2] = PR[GP1:90,2] + 0.325;
   1:L PR[91] 10mm/sec CNT100;
   1:  PR[GP1:91,1] = PR[GP1:90,1] + 26.494;
   1:  PR[GP1:91,2] = PR[GP1:90,2] + 0.921;
   1:L PR[91] 10mm/sec CNT100;
   1:  PR[GP1:91,1] = PR[GP1:90,1] + 25.272;
   1:  PR[GP1:91,2] = PR[GP1:90,2] + 3.060;
   1:L PR[91] 10mm/sec CNT100;
   1:  PR[GP1:91,1] = PR[GP1:90,1] + 24.587;
   1:  PR[GP1:91,2] = PR[GP1:90,2] + 4.204;
   1:L PR[91] 10mm/sec CNT100;
   1:  PR[GP1:91,1] = PR[GP1:90,1] + 23.600;
   1:  PR[GP1:91,2] = PR[GP1:90,2] + 5.354;
   1:L PR[91] 10mm/sec CNT100;
   1:  PR[GP1:91,1] = PR[GP1:90,1] + 22.142;
   1:  PR[GP1:91,2] = PR[GP1:90,2] + 6.996;
   1:L PR[91] 10mm/sec CNT100;
   1:  PR[GP1:91,1] = PR[GP1:90,1] + 21.487;
   1:  PR[GP1:91,2] = PR[GP1:90,2] + 7.516;
   1:L PR[91] 10mm/sec CNT100;
   1:  PR[GP1:91,1] = PR[GP1:90,1] + 19.300;
   1:  PR[GP1:91,2] = PR[GP1:90,2] + 9.200;
   1:L PR[91] 10mm/sec CNT100;
   1:  PR[GP1:91,1] = PR[GP1:90,1] + 16.175;
   1:  PR[GP1:91,2] = PR[GP1:90,2] + 10.771;
   1:L PR[91] 10mm/sec CNT100;
   1:  PR[GP1:91,1] = PR[GP1:90,1] + 12.886;
   1:  PR[GP1:91,2] = PR[GP1:90,2] + 11.675;
   1:L PR[91] 10mm/sec CNT100;
   1:  PR[GP1:91,1] = PR[GP1:90,1] + 9.463;
   1:  PR[GP1:91,2] = PR[GP1:90,2] + 11.925;
   1:L PR[91] 10mm/sec CNT100;
   1:  PR[GP1:91,1] = PR[GP1:90,1] + 6.130;
   1:  PR[GP1:91,2] = PR[GP1:90,2] + 11.482;
   1:L PR[91] 10mm/sec CNT100;
   1:  PR[GP1:91,1] = PR[GP1:90,1] + 4.638;
   1:  PR[GP1:91,2] = PR[GP1:90,2] + 11.112;
   1:L PR[91] 10mm/sec CNT100;
   1:  PR[GP1:91,1] = PR[GP1:90,1] + 3.452;
   1:  PR[GP1:91,2] = PR[GP1:90,2] + 11.046;
   1:L PR[91] 10mm/sec CNT100;
   1:  PR[GP1:91,1] = PR[GP1:90,1] + 1.614;
   1:  PR[GP1:91,2] = PR[GP1:90,2] + 11.320;
   1:L PR[91] 10mm/sec CNT100;
   1:  PR[GP1:91,1] = PR[GP1:90,1] + 0.608;
   1:  PR[GP1:91,2] = PR[GP1:90,2] + 11.435;
   1:L PR[91] 10mm/sec CNT100;
   1:  PR[GP1:91,1] = PR[GP1:90,1] + -0.081;
   1:  PR[GP1:91,2] = PR[GP1:90,2] + 11.438;
   1:L PR[91] 10mm/sec CNT100;
   1:  PR[GP1:91,1] = PR[GP1:90,1] + -2.695;
   1:  PR[GP1:91,2] = PR[GP1:90,2] + 11.512;
   1:L PR[91] 10mm/sec CNT100;
   1:  PR[GP1:91,1] = PR[GP1:90,1] + -4.010;
   1:  PR[GP1:91,2] = PR[GP1:90,2] + 11.518;
   1:L PR[91] 10mm/sec CNT100;
   1:  PR[GP1:91,1] = PR[GP1:90,1] + -4.215;
   1:  PR[GP1:91,2] = PR[GP1:90,2] + 11.498;
   1:L PR[91] 10mm/sec CNT100;
   1:  PR[GP1:91,1] = PR[GP1:90,1] + -7.831;
   1:  PR[GP1:91,2] = PR[GP1:90,2] + 10.896;
   1:L PR[91] 10mm/sec CNT100;
   1:  PR[GP1:91,1] = PR[GP1:90,1] + -8.630;
   1:  PR[GP1:91,2] = PR[GP1:90,2] + 10.722;
   1:L PR[91] 10mm/sec CNT100;
   1:  PR[GP1:91,1] = PR[GP1:90,1] + -9.671;
   1:  PR[GP1:91,2] = PR[GP1:90,2] + 10.357;
   1:L PR[91] 10mm/sec CNT100;
   1:  PR[GP1:91,1] = PR[GP1:90,1] + -12.074;
   1:  PR[GP1:91,2] = PR[GP1:90,2] + 9.474;
   1:L PR[91] 10mm/sec CNT100;
   1:  PR[GP1:91,1] = PR[GP1:90,1] + -13.386;
   1:  PR[GP1:91,2] = PR[GP1:90,2] + 8.796;
   1:L PR[91] 10mm/sec CNT100;
   1:  PR[GP1:91,1] = PR[GP1:90,1] + -14.747;
   1:  PR[GP1:91,2] = PR[GP1:90,2] + 7.945;
   1:L PR[91] 10mm/sec CNT100;
   1:  PR[GP1:91,1] = PR[GP1:90,1] + -16.092;
   1:  PR[GP1:91,2] = PR[GP1:90,2] + 6.980;
   1:L PR[91] 10mm/sec CNT100;
   1:  PR[GP1:91,1] = PR[GP1:90,1] + -18.084;
   1:  PR[GP1:91,2] = PR[GP1:90,2] + 4.981;
   1:L PR[91] 10mm/sec CNT100;
   1:  PR[GP1:91,1] = PR[GP1:90,1] + -19.248;
   1:  PR[GP1:91,2] = PR[GP1:90,2] + 3.329;
   1:L PR[91] 10mm/sec CNT100;
   1:  PR[GP1:91,1] = PR[GP1:90,1] + -19.538;
   1:  PR[GP1:91,2] = PR[GP1:90,2] + 2.823;
   1:L PR[91] 10mm/sec CNT100;
   1:  PR[GP1:91,1] = PR[GP1:90,1] + -20.435;
   1:  PR[GP1:91,2] = PR[GP1:90,2] + 0.955;
   1:L PR[91] 10mm/sec CNT100;
   1:  PR[GP1:91,1] = PR[GP1:90,1] + -21.117;
   1:  PR[GP1:91,2] = PR[GP1:90,2] + -1.400;
   1:L PR[91] 10mm/sec CNT100;
   1:  PR[GP1:91,1] = PR[GP1:90,1] + -21.297;
   1:  PR[GP1:91,2] = PR[GP1:90,2] + -3.092;
   1:L PR[91] 10mm/sec CNT100;
   1:  PR[GP1:91,1] = PR[GP1:90,1] + -21.158;
   1:  PR[GP1:91,2] = PR[GP1:90,2] + -4.636;
   1:L PR[91] 10mm/sec CNT100;
   1:  PR[GP1:91,1] = PR[GP1:90,1] + -21.138;
   1:  PR[GP1:91,2] = PR[GP1:90,2] + -5.289;
   1:L PR[91] 10mm/sec CNT100;
   1:  PR[GP1:91,1] = PR[GP1:90,1] + -20.511;
   1:  PR[GP1:91,2] = PR[GP1:90,2] + -7.867;
   1:L PR[91] 10mm/sec CNT100;
   1:  PR[GP1:91,1] = PR[GP1:90,1] + -20.212;
   1:  PR[GP1:91,2] = PR[GP1:90,2] + -8.828;
   1:L PR[91] 10mm/sec CNT100;
   1:  PR[GP1:91,1] = PR[GP1:90,1] + -19.379;
   1:  PR[GP1:91,2] = PR[GP1:90,2] + -10.810;
   1:L PR[91] 10mm/sec CNT100;
   1:  PR[GP1:91,1] = PR[GP1:90,1] + -18.497;
   1:  PR[GP1:91,2] = PR[GP1:90,2] + -12.272;
   1:L PR[91] 10mm/sec CNT100;
   1:  PR[GP1:91,1] = PR[GP1:90,1] + -17.481;
   1:  PR[GP1:91,2] = PR[GP1:90,2] + -13.848;
   1:L PR[91] 10mm/sec CNT100;
   1:  PR[GP1:91,1] = PR[GP1:90,1] + -16.447;
   1:  PR[GP1:91,2] = PR[GP1:90,2] + -15.014;
   1:L PR[91] 10mm/sec CNT100;
   1:  PR[GP1:91,1] = PR[GP1:90,1] + -13.280;
   1:  PR[GP1:91,2] = PR[GP1:90,2] + -17.609;
   1:  PR[GP1:91,3] = PR[GP1:90,3] + 47.300;
   1:L PR[91] 10mm/sec CNT100;
   1:  PR[GP1:91,1] = PR[GP1:90,1] + -12.805;
   1:  PR[GP1:91,2] = PR[GP1:90,2] + -18.018;
   1:L PR[91] 10mm/sec CNT100;
   1:  PR[GP1:91,1] = PR[GP1:90,1] + -9.965;
   1:  PR[GP1:91,2] = PR[GP1:90,2] + -19.955;
   1:L PR[91] 10mm/sec CNT100;
   1:  PR[GP1:91,1] = PR[GP1:90,1] + -8.798;
   1:  PR[GP1:91,2] = PR[GP1:90,2] + -20.833;
   1:L PR[91] 10mm/sec CNT100;
   1:  PR[GP1:91,1] = PR[GP1:90,1] + -8.484;
   1:  PR[GP1:91,2] = PR[GP1:90,2] + -21.044;
   1:L PR[91] 10mm/sec CNT100;
   1:  PR[GP1:91,1] = PR[GP1:90,1] + -4.716;
   1:  PR[GP1:91,2] = PR[GP1:90,2] + -22.936;
   1:L PR[91] 10mm/sec CNT100;
   1:  PR[GP1:91,1] = PR[GP1:90,1] + -2.954;
   1:  PR[GP1:91,2] = PR[GP1:90,2] + -23.704;
   1:L PR[91] 10mm/sec CNT100;
   1:  PR[GP1:91,1] = PR[GP1:90,1] + -0.321;
   1:  PR[GP1:91,2] = PR[GP1:90,2] + -24.488;
   1:L PR[91] 10mm/sec CNT100;
   1:  PR[GP1:91,1] = PR[GP1:90,1] + 3.086;
   1:  PR[GP1:91,2] = PR[GP1:90,2] + -25.288;
   1:L PR[91] 10mm/sec CNT100;
   1:  PR[GP1:91,1] = PR[GP1:90,1] + 4.288;
   1:  PR[GP1:91,2] = PR[GP1:90,2] + -25.418;
   1:L PR[91] 10mm/sec CNT100;
   1:  PR[GP1:91,1] = PR[GP1:90,1] + 8.595;
   1:  PR[GP1:91,2] = PR[GP1:90,2] + -25.597;
   1:L PR[91] 10mm/sec CNT100;
   1:  PR[GP1:91,1] = PR[GP1:90,1] + 9.137;
   1:  PR[GP1:91,2] = PR[GP1:90,2] + -25.649;
   1:L PR[91] 10mm/sec CNT100;
   1:  PR[GP1:91,1] = PR[GP1:90,1] + 9.569;
   1:  PR[GP1:91,2] = PR[GP1:90,2] + -25.663;
   1:L PR[91] 10mm/sec CNT100;
   1:  PR[GP1:91,1] = PR[GP1:90,1] + 10.959;
   1:  PR[GP1:91,2] = PR[GP1:90,2] + -25.790;
   1:L PR[91] 10mm/sec CNT100;
   1:  PR[GP1:91,1] = PR[GP1:90,1] + 12.787;
   1:  PR[GP1:91,2] = PR[GP1:90,2] + -25.840;
   1:L PR[91] 10mm/sec CNT100;
   1:  PR[GP1:91,1] = PR[GP1:90,1] + 13.430;
   1:  PR[GP1:91,2] = PR[GP1:90,2] + -25.794;
   1:L PR[91] 10mm/sec CNT100;
   1:  PR[GP1:91,1] = PR[GP1:90,1] + 15.745;
   1:  PR[GP1:91,2] = PR[GP1:90,2] + -25.499;
   1:L PR[91] 10mm/sec CNT100;
   1:  PR[GP1:91,1] = PR[GP1:90,1] + 18.273;
   1:  PR[GP1:91,2] = PR[GP1:90,2] + -24.802;
   1:L PR[91] 10mm/sec CNT100;
   1:  PR[GP1:91,1] = PR[GP1:90,1] + 18.698;
   1:  PR[GP1:91,2] = PR[GP1:90,2] + -24.644;
   1:L PR[91] 10mm/sec CNT100;
   1:  PR[GP1:91,1] = PR[GP1:90,1] + 20.605;
   1:  PR[GP1:91,2] = PR[GP1:90,2] + -23.766;
   1:L PR[91] 10mm/sec CNT100;
   1:  PR[GP1:91,1] = PR[GP1:90,1] + 21.437;
   1:  PR[GP1:91,2] = PR[GP1:90,2] + -23.276;
   1:L PR[91] 10mm/sec CNT100;
   1:  PR[GP1:91,1] = PR[GP1:90,1] + 22.804;
   1:  PR[GP1:91,2] = PR[GP1:90,2] + -22.335;
   1:L PR[91] 10mm/sec CNT100;
   1:  PR[GP1:91,1] = PR[GP1:90,1] + 23.762;
   1:  PR[GP1:91,2] = PR[GP1:90,2] + -21.506;
   1:L PR[91] 10mm/sec CNT100;
   1:  PR[GP1:91,1] = PR[GP1:90,1] + 24.787;
   1:  PR[GP1:91,2] = PR[GP1:90,2] + -20.495;
   1:L PR[91] 10mm/sec CNT100;
   1:  PR[GP1:91,1] = PR[GP1:90,1] + 25.603;
   1:  PR[GP1:91,2] = PR[GP1:90,2] + -19.468;
   1:L PR[91] 10mm/sec CNT100;
   1:  PR[GP1:91,1] = PR[GP1:90,1] + 26.454;
   1:  PR[GP1:91,2] = PR[GP1:90,2] + -18.262;
   1:L PR[91] 10mm/sec CNT100;
   1:  PR[GP1:91,1] = PR[GP1:90,1] + 26.968;
   1:  PR[GP1:91,2] = PR[GP1:90,2] + -17.299;
   1:L PR[91] 10mm/sec CNT100;
   1:  PR[GP1:91,1] = PR[GP1:90,1] + 27.724;
   1:  PR[GP1:91,2] = PR[GP1:90,2] + -15.706;
   1:L PR[91] 10mm/sec CNT100;
   1:  PR[GP1:91,1] = PR[GP1:90,1] + 27.923;
   1:  PR[GP1:91,2] = PR[GP1:90,2] + -15.104;
   1:L PR[91] 10mm/sec CNT100;
   1:  PR[GP1:91,1] = PR[GP1:90,1] + 28.548;
   1:  PR[GP1:91,2] = PR[GP1:90,2] + -12.952;
   1:L PR[91] 10mm/sec CNT100;
   1:  PR[GP1:91,1] = PR[GP1:90,1] + 28.961;
   1:  PR[GP1:91,2] = PR[GP1:90,2] + -10.178;
   1:L PR[91] 10mm/sec CNT100;
   1:  PR[GP1:91,1] = PR[GP1:90,1] + 28.872;
   1:  PR[GP1:91,2] = PR[GP1:90,2] + -7.260;
   1:L PR[91] 10mm/sec CNT100;
   1:  PR[GP1:91,1] = PR[GP1:90,1] + 28.338;
   1:  PR[GP1:91,2] = PR[GP1:90,2] + -4.394;
   1:L PR[91] 10mm/sec CNT100;
   1:  PR[GP1:91,1] = PR[GP1:90,1] + 28.154;
   1:  PR[GP1:91,2] = PR[GP1:90,2] + -3.290;
   1:L PR[91] 10mm/sec CNT100;
   1:  PR[GP1:91,1] = PR[GP1:90,1] + 26.806;
   1:  PR[GP1:91,2] = PR[GP1:90,2] + 0.437;
   1:L PR[91] 10mm/sec CNT100;
   1:  PR[GP1:91,1] = PR[GP1:90,1] + 26.404;
   1:  PR[GP1:91,2] = PR[GP1:90,2] + 1.127;
   1:L PR[91] 10mm/sec CNT100;
   1:  PR[GP1:91,1] = PR[GP1:90,1] + 25.207;
   1:  PR[GP1:91,2] = PR[GP1:90,2] + 3.087;
   1:L PR[91] 10mm/sec CNT100;
   1:  PR[GP1:91,1] = PR[GP1:90,1] + 24.800;
   1:  PR[GP1:91,2] = PR[GP1:90,2] + 3.791;
   1:L PR[91] 10mm/sec CNT100;
   1:  PR[GP1:91,1] = PR[GP1:90,1] + 23.087;
   1:  PR[GP1:91,2] = PR[GP1:90,2] + 5.786;
   1:L PR[91] 10mm/sec CNT100;
   1:  PR[GP1:91,1] = PR[GP1:90,1] + 22.351;
   1:  PR[GP1:91,2] = PR[GP1:90,2] + 6.614;
   1:L PR[91] 10mm/sec CNT100;
   1:  PR[GP1:91,1] = PR[GP1:90,1] + 20.866;
   1:  PR[GP1:91,2] = PR[GP1:90,2] + 7.795;
   1:L PR[91] 10mm/sec CNT100;
   1:  PR[GP1:91,1] = PR[GP1:90,1] + 19.493;
   1:  PR[GP1:91,2] = PR[GP1:90,2] + 8.852;
   1:L PR[91] 10mm/sec CNT100;
   1:  PR[GP1:91,1] = PR[GP1:90,1] + 18.131;
   1:  PR[GP1:91,2] = PR[GP1:90,2] + 9.558;
   1:L PR[91] 10mm/sec CNT100;
   1:  PR[GP1:91,1] = PR[GP1:90,1] + 16.343;
   1:  PR[GP1:91,2] = PR[GP1:90,2] + 10.452;
   1:L PR[91] 10mm/sec CNT100;
   1:  PR[GP1:91,1] = PR[GP1:90,1] + 14.463;
   1:  PR[GP1:91,2] = PR[GP1:90,2] + 10.991;
   1:L PR[91] 10mm/sec CNT100;
   1:  PR[GP1:91,1] = PR[GP1:90,1] + 13.005;
   1:  PR[GP1:91,2] = PR[GP1:90,2] + 11.388;
   1:L PR[91] 10mm/sec CNT100;
   1:  PR[GP1:91,1] = PR[GP1:90,1] + 9.579;
   1:  PR[GP1:91,2] = PR[GP1:90,2] + 11.648;
   1:L PR[91] 10mm/sec CNT100;
   1:  PR[GP1:91,1] = PR[GP1:90,1] + 8.545;
   1:  PR[GP1:91,2] = PR[GP1:90,2] + 11.536;
   1:L PR[91] 10mm/sec CNT100;
   1:  PR[GP1:91,1] = PR[GP1:90,1] + 6.219;
   1:  PR[GP1:91,2] = PR[GP1:90,2] + 11.224;
   1:L PR[91] 10mm/sec CNT100;
   1:  PR[GP1:91,1] = PR[GP1:90,1] + 4.959;
   1:  PR[GP1:91,2] = PR[GP1:90,2] + 10.926;
   1:L PR[91] 10mm/sec CNT100;
   1:  PR[GP1:91,1] = PR[GP1:90,1] + 3.841;
   1:  PR[GP1:91,2] = PR[GP1:90,2] + 10.866;
   1:L PR[91] 10mm/sec CNT100;
   1:  PR[GP1:91,1] = PR[GP1:90,1] + 2.394;
   1:  PR[GP1:91,2] = PR[GP1:90,2] + 11.066;
   1:L PR[91] 10mm/sec CNT100;
   1:  PR[GP1:91,1] = PR[GP1:90,1] + 1.499;
   1:  PR[GP1:91,2] = PR[GP1:90,2] + 11.153;
   1:L PR[91] 10mm/sec CNT100;
   1:  PR[GP1:91,1] = PR[GP1:90,1] + 0.316;
   1:  PR[GP1:91,2] = PR[GP1:90,2] + 11.159;
   1:L PR[91] 10mm/sec CNT100;
   1:  PR[GP1:91,1] = PR[GP1:90,1] + -3.211;
   1:  PR[GP1:91,2] = PR[GP1:90,2] + 11.258;
   1:L PR[91] 10mm/sec CNT100;
   1:  PR[GP1:91,1] = PR[GP1:90,1] + -4.014;
   1:  PR[GP1:91,2] = PR[GP1:90,2] + 11.136;
   1:L PR[91] 10mm/sec CNT100;
   1:  PR[GP1:91,1] = PR[GP1:90,1] + -7.223;
   1:  PR[GP1:91,2] = PR[GP1:90,2] + 10.602;
   1:L PR[91] 10mm/sec CNT100;
   1:  PR[GP1:91,1] = PR[GP1:90,1] + -7.678;
   1:  PR[GP1:91,2] = PR[GP1:90,2] + 10.503;
   1:L PR[91] 10mm/sec CNT100;
   1:  PR[GP1:91,1] = PR[GP1:90,1] + -11.292;
   1:  PR[GP1:91,2] = PR[GP1:90,2] + 9.185;
   1:L PR[91] 10mm/sec CNT100;
   1:  PR[GP1:91,1] = PR[GP1:90,1] + -12.270;
   1:  PR[GP1:91,2] = PR[GP1:90,2] + 8.680;
   1:L PR[91] 10mm/sec CNT100;
   1:  PR[GP1:91,1] = PR[GP1:90,1] + -14.078;
   1:  PR[GP1:91,2] = PR[GP1:90,2] + 7.550;
   1:L PR[91] 10mm/sec CNT100;
   1:  PR[GP1:91,1] = PR[GP1:90,1] + -15.162;
   1:  PR[GP1:91,2] = PR[GP1:90,2] + 6.772;
   1:L PR[91] 10mm/sec CNT100;
   1:  PR[GP1:91,1] = PR[GP1:90,1] + -16.273;
   1:  PR[GP1:91,2] = PR[GP1:90,2] + 5.667;
   1:L PR[91] 10mm/sec CNT100;
   1:  PR[GP1:91,1] = PR[GP1:90,1] + -17.265;
   1:  PR[GP1:91,2] = PR[GP1:90,2] + 4.652;
   1:L PR[91] 10mm/sec CNT100;
   1:  PR[GP1:91,1] = PR[GP1:90,1] + -18.234;
   1:  PR[GP1:91,2] = PR[GP1:90,2] + 3.277;
   1:L PR[91] 10mm/sec CNT100;
   1:  PR[GP1:91,1] = PR[GP1:90,1] + -18.770;
   1:  PR[GP1:91,2] = PR[GP1:90,2] + 2.341;
   1:L PR[91] 10mm/sec CNT100;
   1:  PR[GP1:91,1] = PR[GP1:90,1] + -19.523;
   1:  PR[GP1:91,2] = PR[GP1:90,2] + 0.772;
   1:L PR[91] 10mm/sec CNT100;
   1:  PR[GP1:91,1] = PR[GP1:90,1] + -20.250;
   1:  PR[GP1:91,2] = PR[GP1:90,2] + -1.757;
   1:L PR[91] 10mm/sec CNT100;
   1:  PR[GP1:91,1] = PR[GP1:90,1] + -20.400;
   1:  PR[GP1:91,2] = PR[GP1:90,2] + -3.169;
   1:L PR[91] 10mm/sec CNT100;
   1:  PR[GP1:91,1] = PR[GP1:90,1] + -20.283;
   1:  PR[GP1:91,2] = PR[GP1:90,2] + -4.467;
   1:L PR[91] 10mm/sec CNT100;
   1:  PR[GP1:91,1] = PR[GP1:90,1] + -20.247;
   1:  PR[GP1:91,2] = PR[GP1:90,2] + -5.611;
   1:L PR[91] 10mm/sec CNT100;
   1:  PR[GP1:91,1] = PR[GP1:90,1] + -19.706;
   1:  PR[GP1:91,2] = PR[GP1:90,2] + -7.857;
   1:L PR[91] 10mm/sec CNT100;
   1:  PR[GP1:91,1] = PR[GP1:90,1] + -19.261;
   1:  PR[GP1:91,2] = PR[GP1:90,2] + -9.286;
   1:L PR[91] 10mm/sec CNT100;
   1:  PR[GP1:91,1] = PR[GP1:90,1] + -18.561;
   1:  PR[GP1:91,2] = PR[GP1:90,2] + -10.951;
   1:L PR[91] 10mm/sec CNT100;
   1:  PR[GP1:91,1] = PR[GP1:90,1] + -17.376;
   1:  PR[GP1:91,2] = PR[GP1:90,2] + -12.916;
   1:L PR[91] 10mm/sec CNT100;
   1:  PR[GP1:91,1] = PR[GP1:90,1] + -16.579;
   1:  PR[GP1:91,2] = PR[GP1:90,2] + -14.152;
   1:L PR[91] 10mm/sec CNT100;
